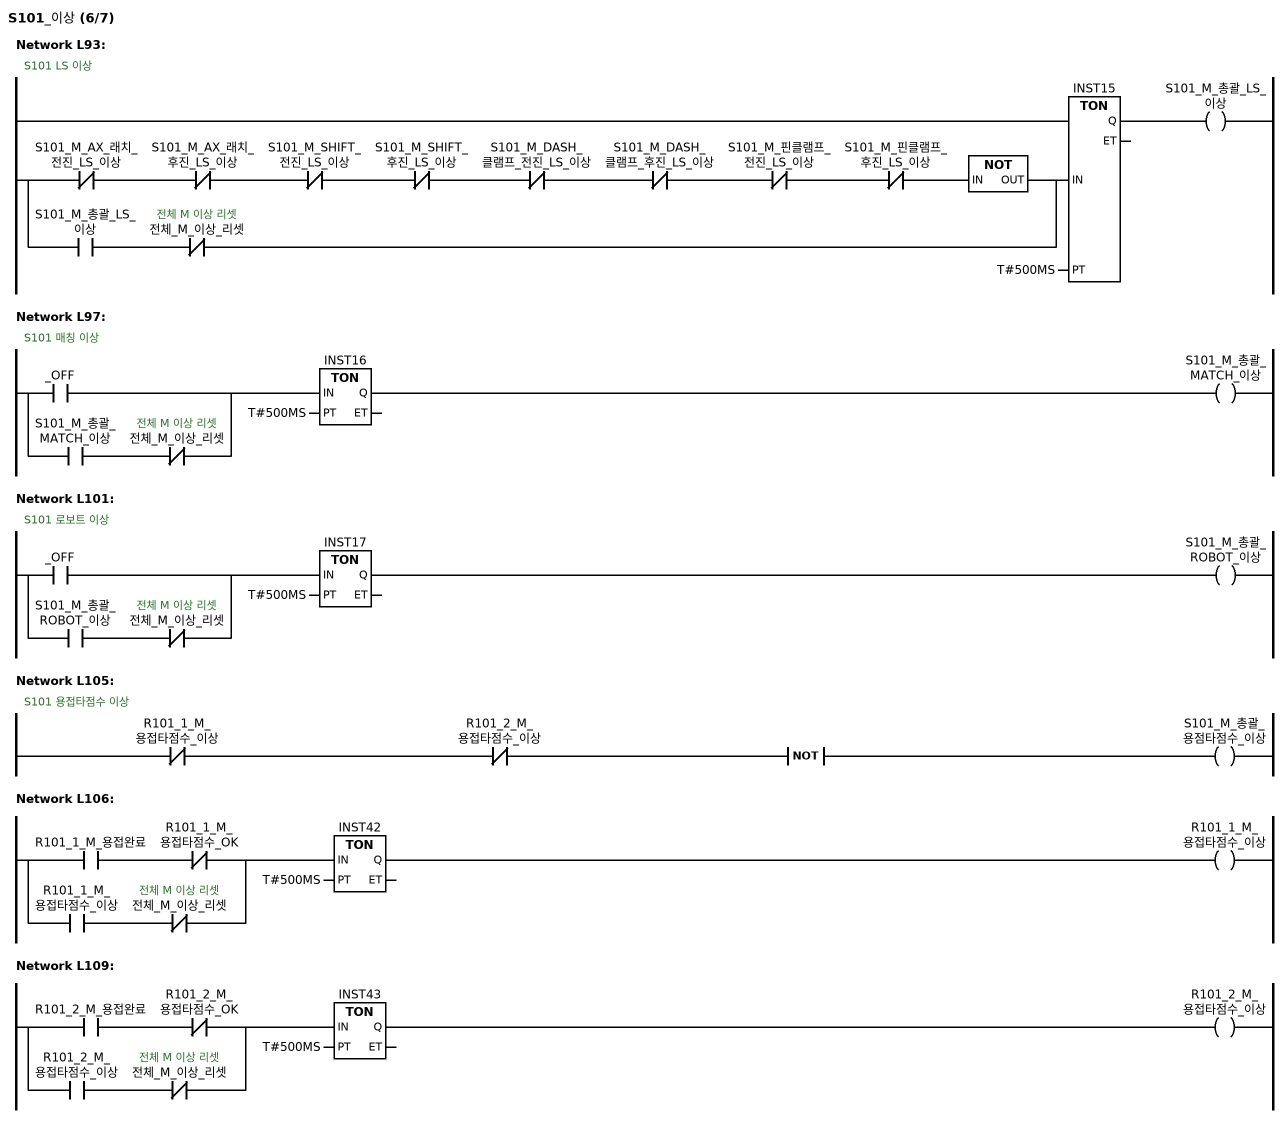
(* [picture p96: S101_이상 rungs L93-L109] *)
(* S101 LS 이상 *)
(* Rung L93 *)
INST15(IN := (NOT (NOT S101_M_AX_래치_전진_LS_이상 AND NOT S101_M_AX_래치_후진_LS_이상 AND NOT S101_M_SHIFT_전진_LS_이상 AND NOT S101_M_SHIFT_후진_LS_이상 AND NOT S101_M_DASH_클램프_전진_LS_이상 AND NOT S101_M_DASH_클램프_후진_LS_이상 AND NOT S101_M_핀클램프_전진_LS_이상 AND NOT S101_M_핀클램프_후진_LS_이상)) OR (S101_M_총괄_LS_이상 AND NOT 전체_M_이상_리셋), PT := T#500MS);
S101_M_총괄_LS_이상 := INST15.Q;
(* S101 매칭 이상 *)
(* Rung L97 *)
INST16(IN := _OFF OR (S101_M_총괄_MATCH_이상 AND NOT 전체_M_이상_리셋), PT := T#500MS);
S101_M_총괄_MATCH_이상 := INST16.Q;
(* S101 로보트 이상 *)
(* Rung L101 *)
INST17(IN := _OFF OR (S101_M_총괄_ROBOT_이상 AND NOT 전체_M_이상_리셋), PT := T#500MS);
S101_M_총괄_ROBOT_이상 := INST17.Q;
(* S101 용접타점수 이상 *)
(* Rung L105 *)
S101_M_총괄_용점타점수_이상 := NOT (NOT R101_1_M_용접타점수_이상 AND NOT R101_2_M_용접타점수_이상);
(* Rung L106 *)
INST42(IN := (R101_1_M_용접완료 AND NOT R101_1_M_용접타점수_OK) OR (R101_1_M_용접타점수_이상 AND NOT 전체_M_이상_리셋), PT := T#500MS);
R101_1_M_용접타점수_이상 := INST42.Q;
(* Rung L109 *)
INST43(IN := (R101_2_M_용접완료 AND NOT R101_2_M_용접타점수_OK) OR (R101_2_M_용접타점수_이상 AND NOT 전체_M_이상_리셋), PT := T#500MS);
R101_2_M_용접타점수_이상 := INST43.Q;

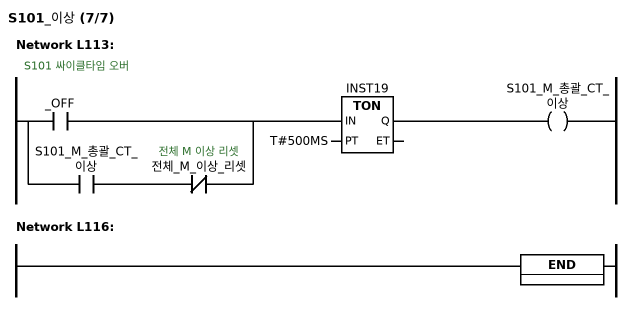
(* S101 싸이클타임 오버 *)
(* Rung L113 *)
INST19(IN := _OFF OR (S101_M_총괄_CT_이상 AND NOT 전체_M_이상_리셋), PT := T#500MS);
S101_M_총괄_CT_이상 := INST19.Q;
(* Rung L116 *)
END();
END_PROGRAM

PROGRAM S102_유틸리티 (* task: 스캔 프로그램 *)
VAR_EXTERNAL
    AWAYS_ON : BOOL; (* AT %MW3.1 *)
    MCP_PBL_102_자동_운전 : BOOL; (* AT %MW87630.7 *) (* 입력 접점 07 *)
    MCP_PBL_운전준비_ON : BOOL; (* AT %MW87630.0 *) (* 입력 접점 00 *)
    MCP_SSP_102_수동_선택 : BOOL; (* AT %MW87630.5 *) (* 입력 접점 05 *)
    MCP_SSP_102_자동_선택 : BOOL; (* AT %MW87630.6 *) (* 입력 접점 06 *)
    R102_1_1_M_I_RB_2차_작업완료 : BOOL; (* AT %MW20091.3 *)
    R102_1_1_M_I_RB_간섭무_1 : BOOL; (* AT %MW20092.0 *)
    R102_1_1_M_I_RB_원위치 : BOOL; (* AT %MW20090.3 *)
    R102_1_1_M_SEQ : WORD; (* AT %MW10040 *) (* R102_1_1_M_SEQ *)
    R102_1_1_M_STN_차종_NONE : BOOL; (* AT %MW1502.3 *)
    R102_1_1_M_STN_차종_ON : BOOL; (* AT %MW1502.2 *)
    R102_1_1_M_차종1_AX : BOOL; (* AT %MW10041.0 *) (* R102_1_1_M_차종1_AX *)
    R102_1_1_M_차종1_B : BOOL; (* AT %MW10041.1 *) (* R102_1_1_M_차종1_B *)
    R102_1_1_M_차종1_C : BOOL; (* AT %MW10041.2 *) (* R102_1_1_M_차종1_C *)
    R102_1_1_M_차종1_D : BOOL; (* AT %MW10041.3 *) (* R102_1_1_M_차종1_D *)
    R102_1_1_M_차종1_E : BOOL; (* AT %MW10041.4 *) (* R102_1_1_M_차종1_E *)
    R102_1_1_M_차종1_F : BOOL; (* AT %MW10041.5 *) (* R102_1_1_M_차종1_F *)
    R102_1_1_M_차종1_G : BOOL; (* AT %MW10041.6 *) (* R102_1_1_M_차종1_G *)
    R102_1_1_M_차종1_H : BOOL; (* AT %MW10041.7 *) (* R102_1_1_M_차종1_H *)
    R102_1_1_M_차종2_3DR : BOOL; (* AT %MW10041.8 *) (* R102_1_1_M_차종2_3DR *)
    R102_1_1_M_차종2_4DR : BOOL; (* AT %MW10041.9 *) (* R102_1_1_M_차종2_4DR *)
    R102_1_1_M_차종2_5DR : BOOL; (* AT %MW10041.10 *) (* R102_1_1_M_차종2_5DR *)
    R102_1_1_M_차종2_SP1 : BOOL; (* AT %MW10041.12 *) (* R102_1_1_M_차종2_SP1 *)
    R102_1_1_M_차종2_SP2 : BOOL; (* AT %MW10041.13 *) (* R102_1_1_M_차종2_SP2 *)
    R102_1_1_M_차종2_WGN : BOOL; (* AT %MW10041.11 *) (* R102_1_1_M_차종2_WGN *)
    R102_1_1_M_차종3_LHD : BOOL; (* AT %MW10041.14 *) (* R102_1_1_M_차종3_LHD *)
    R102_1_1_M_차종3_RHD : BOOL; (* AT %MW10041.15 *) (* R102_1_1_M_차종3_RHD *)
    R102_1_1_M_차종4_EEC : BOOL; (* AT %MW10042.3 *) (* R102_1_1_M_차종4_EEC *)
    R102_1_1_M_차종4_SP1 : BOOL; (* AT %MW10042.8 *) (* R102_1_1_M_차종4_SP1 *)
    R102_1_1_M_차종4_SP2 : BOOL; (* AT %MW10042.9 *) (* R102_1_1_M_차종4_SP2 *)
    R102_1_1_M_차종4_SP3 : BOOL; (* AT %MW10042.11 *) (* R102_1_1_M_차종4_SP3 *)
    R102_1_1_M_차종4_SP4 : BOOL; (* AT %MW10042.12 *) (* R102_1_1_M_차종4_SP4 *)
    R102_1_1_M_차종4_SP5 : BOOL; (* AT %MW10042.13 *) (* R102_1_1_M_차종4_SP5 *)
    R102_1_1_M_차종4_SP6 : BOOL; (* AT %MW10042.14 *) (* R102_1_1_M_차종4_SP6 *)
    R102_1_1_M_차종4_SP7 : BOOL; (* AT %MW10042.15 *) (* R102_1_1_M_차종4_SP7 *)
    R102_1_1_M_차종4_내수 : BOOL; (* AT %MW10042.0 *) (* R102_1_1_M_차종4_내수 *)
    R102_1_1_M_차종4_러시아 : BOOL; (* AT %MW10042.10 *) (* R102_1_1_M_차종4_러시아 *)
    R102_1_1_M_차종4_북미 : BOOL; (* AT %MW10042.2 *) (* R102_1_1_M_차종4_북미 *)
    R102_1_1_M_차종4_브라질 : BOOL; (* AT %MW10042.7 *) (* R102_1_1_M_차종4_브라질 *)
    R102_1_1_M_차종4_수출 : BOOL; (* AT %MW10042.1 *) (* R102_1_1_M_차종4_수출 *)
    R102_1_1_M_차종4_중국 : BOOL; (* AT %MW10042.6 *) (* R102_1_1_M_차종4_중국 *)
    R102_1_1_M_차종4_중동 : BOOL; (* AT %MW10042.5 *) (* R102_1_1_M_차종4_중동 *)
    R102_1_1_M_차종4_호주 : BOOL; (* AT %MW10042.4 *) (* R102_1_1_M_차종4_호주 *)
    R102_1_1_M_차종5_AT : BOOL; (* AT %MW10043.1 *) (* R102_1_1_M_차종5_AT *)
    R102_1_1_M_차종5_MT : BOOL; (* AT %MW10043.0 *) (* R102_1_1_M_차종5_MT *)
    R102_1_1_M_차종5_SP1 : BOOL; (* AT %MW10043.2 *) (* R102_1_1_M_차종5_SP1 *)
    R102_1_1_M_차종6_DSROOF : BOOL; (* AT %MW10043.6 *) (* R102_1_1_M_차종6_DSROOF *)
    R102_1_1_M_차종6_SP1 : BOOL; (* AT %MW10043.7 *) (* R102_1_1_M_차종6_SP1 *)
    R102_1_1_M_차종6_썬루프 : BOOL; (* AT %MW10043.4 *) (* R102_1_1_M_차종6_썬루프 *)
    R102_1_1_M_차종6_일반루프 : BOOL; (* AT %MW10043.3 *) (* R102_1_1_M_차종6_일반루프 *)
    R102_1_1_M_차종6_파노라마루프 : BOOL; (* AT %MW10043.5 *) (* R102_1_1_M_차종6_파노라마루프 *)
    R102_1_1_M_차종7_DSL : BOOL; (* AT %MW10043.9 *) (* R102_1_1_M_차종7_DSL *)
    R102_1_1_M_차종7_GSL : BOOL; (* AT %MW10043.8 *) (* R102_1_1_M_차종7_GSL *)
    R102_1_1_M_차종7_SP1 : BOOL; (* AT %MW10043.10 *) (* R102_1_1_M_차종7_SP1 *)
    R102_1_1_M_차종7_SP2 : BOOL; (* AT %MW10043.11 *) (* R102_1_1_M_차종7_SP2 *)
    R102_1_1_M_차종7_SP3 : BOOL; (* AT %MW10043.12 *) (* R102_1_1_M_차종7_SP3 *)
    R102_1_1_M_차종7_SP4 : BOOL; (* AT %MW10043.13 *) (* R102_1_1_M_차종7_SP4 *)
    R102_1_1_M_차종7_SP5 : BOOL; (* AT %MW10043.14 *) (* R102_1_1_M_차종7_SP5 *)
    R102_1_1_M_차종7_SP6 : BOOL; (* AT %MW10043.15 *) (* R102_1_1_M_차종7_SP6 *)
    R102_1_1_M_차종8_2WD : BOOL; (* AT %MW10044.0 *) (* R102_1_1_M_차종8_2WD *)
    R102_1_1_M_차종8_4WD : BOOL; (* AT %MW10044.1 *) (* R102_1_1_M_차종8_4WD *)
    R102_1_1_M_차종8_SP1 : BOOL; (* AT %MW10044.2 *) (* R102_1_1_M_차종8_SP1 *)
    R102_1_1_M_차종9_MPI : BOOL; (* AT %MW10044.3 *) (* R102_1_1_M_차종9_MPI *)
    R102_1_1_M_차종9_SP1 : BOOL; (* AT %MW10044.5 *) (* R102_1_1_M_차종9_SP1 *)
    R102_1_1_M_차종9_SP10 : BOOL; (* AT %MW10044.14 *) (* R102_1_1_M_차종9_SP10 *)
    R102_1_1_M_차종9_SP11 : BOOL; (* AT %MW10044.15 *) (* R102_1_1_M_차종9_SP11 *)
    R102_1_1_M_차종9_SP2 : BOOL; (* AT %MW10044.6 *) (* R102_1_1_M_차종9_SP2 *)
    R102_1_1_M_차종9_SP3 : BOOL; (* AT %MW10044.7 *) (* R102_1_1_M_차종9_SP3 *)
    R102_1_1_M_차종9_SP4 : BOOL; (* AT %MW10044.8 *) (* R102_1_1_M_차종9_SP4 *)
    R102_1_1_M_차종9_SP5 : BOOL; (* AT %MW10044.9 *) (* R102_1_1_M_차종9_SP5 *)
    R102_1_1_M_차종9_SP6 : BOOL; (* AT %MW10044.10 *) (* R102_1_1_M_차종9_SP6 *)
    R102_1_1_M_차종9_SP7 : BOOL; (* AT %MW10044.11 *) (* R102_1_1_M_차종9_SP7 *)
    R102_1_1_M_차종9_SP8 : BOOL; (* AT %MW10044.12 *) (* R102_1_1_M_차종9_SP8 *)
    R102_1_1_M_차종9_SP9 : BOOL; (* AT %MW10044.13 *) (* R102_1_1_M_차종9_SP9 *)
    R102_1_1_M_차종9_T_GDI : BOOL; (* AT %MW10044.4 *) (* R102_1_1_M_차종9_T_GDI *)
    R102_1_1_M_차종_OPT1_R_RACK_무 : BOOL; (* AT %MW10045.3 *) (* R102_1_1_M_차종_OPT1_R_RACK_무 *)
    R102_1_1_M_차종_OPT1_R_RACK_유 : BOOL; (* AT %MW10045.2 *) (* R102_1_1_M_차종_OPT1_R_RACK_유 *)
    R102_1_1_M_차종_OPT1_SP1 : BOOL; (* AT %MW10045.10 *) (* R102_1_1_M_차종_OPT1_SP1 *)
    R102_1_1_M_차종_OPT1_SP2 : BOOL; (* AT %MW10045.11 *) (* R102_1_1_M_차종_OPT1_SP2 *)
    R102_1_1_M_차종_OPT1_SP3 : BOOL; (* AT %MW10045.12 *) (* R102_1_1_M_차종_OPT1_SP3 *)
    R102_1_1_M_차종_OPT1_SP4 : BOOL; (* AT %MW10045.13 *) (* R102_1_1_M_차종_OPT1_SP4 *)
    R102_1_1_M_차종_OPT1_SP5 : BOOL; (* AT %MW10045.14 *) (* R102_1_1_M_차종_OPT1_SP5 *)
    R102_1_1_M_차종_OPT1_SP6 : BOOL; (* AT %MW10045.15 *) (* R102_1_1_M_차종_OPT1_SP6 *)
    R102_1_1_M_차종_OPT1_S_REP_EATER_무 : BOOL; (* AT %MW10045.7 *) (* R102_1_1_M_차종_OPT1_S_REP_EATER_무 *)
    R102_1_1_M_차종_OPT1_S_REP_EATER_유 : BOOL; (* AT %MW10045.6 *) (* R102_1_1_M_차종_OPT1_S_REP_EATER_유 *)
    R102_1_1_M_차종_OPT1_VAN_무 : BOOL; (* AT %MW10045.9 *) (* R102_1_1_M_차종_OPT1_VAN_무 *)
    R102_1_1_M_차종_OPT1_VAN_유 : BOOL; (* AT %MW10045.8 *) (* R102_1_1_M_차종_OPT1_VAN_유 *)
    R102_1_1_M_차종_OPT1_슬라이딩_무 : BOOL; (* AT %MW10045.1 *) (* R102_1_1_M_차종_OPT1_슬라이딩_무 *)
    R102_1_1_M_차종_OPT1_슬라이딩_유 : BOOL; (* AT %MW10045.0 *) (* R102_1_1_M_차종_OPT1_슬라이딩_유 *)
    R102_1_1_M_차종_OPT1_폴딩_무 : BOOL; (* AT %MW10045.5 *) (* R102_1_1_M_차종_OPT1_폴딩_무 *)
    R102_1_1_M_차종_OPT1_폴딩_유 : BOOL; (* AT %MW10045.4 *) (* R102_1_1_M_차종_OPT1_폴딩_유 *)
    R102_1_M_I_RB_간섭무_1 : BOOL; (* AT %MW20082.0 *)
    R102_1_M_I_RB_원위치 : BOOL; (* AT %MW20080.3 *)
    R102_1_M_SEQ : WORD; (* AT %MW10080 *) (* R102_1_M_SEQ *)
    R102_1_M_STN_차종_NONE : BOOL; (* AT %MW1502.5 *)
    R102_1_M_STN_차종_ON : BOOL; (* AT %MW1502.4 *)
    R102_1_M_차종1_AX : BOOL; (* AT %MW10081.0 *) (* R102_1_M_차종1_AX *)
    R102_1_M_차종1_B : BOOL; (* AT %MW10081.1 *) (* R102_1_M_차종1_B *)
    R102_1_M_차종1_C : BOOL; (* AT %MW10081.2 *) (* R102_1_M_차종1_C *)
    R102_1_M_차종1_D : BOOL; (* AT %MW10081.3 *) (* R102_1_M_차종1_D *)
    R102_1_M_차종1_E : BOOL; (* AT %MW10081.4 *) (* R102_1_M_차종1_E *)
    R102_1_M_차종1_F : BOOL; (* AT %MW10081.5 *) (* R102_1_M_차종1_F *)
    R102_1_M_차종1_G : BOOL; (* AT %MW10081.6 *) (* R102_1_M_차종1_G *)
    R102_1_M_차종1_H : BOOL; (* AT %MW10081.7 *) (* R102_1_M_차종1_H *)
    R102_1_M_차종2_3DR : BOOL; (* AT %MW10081.8 *) (* R102_1_M_차종2_3DR *)
    R102_1_M_차종2_4DR : BOOL; (* AT %MW10081.9 *) (* R102_1_M_차종2_4DR *)
    R102_1_M_차종2_5DR : BOOL; (* AT %MW10081.10 *) (* R102_1_M_차종2_5DR *)
    R102_1_M_차종2_SP1 : BOOL; (* AT %MW10081.12 *) (* R102_1_M_차종2_SP1 *)
    R102_1_M_차종2_SP2 : BOOL; (* AT %MW10081.13 *) (* R102_1_M_차종2_SP2 *)
    R102_1_M_차종2_WGN : BOOL; (* AT %MW10081.11 *) (* R102_1_M_차종2_WGN *)
    R102_1_M_차종3_LHD : BOOL; (* AT %MW10081.14 *) (* R102_1_M_차종3_LHD *)
    R102_1_M_차종3_RHD : BOOL; (* AT %MW10081.15 *) (* R102_1_M_차종3_RHD *)
    R102_1_M_차종4_EEC : BOOL; (* AT %MW10082.3 *) (* R102_1_M_차종4_EEC *)
    R102_1_M_차종4_SP1 : BOOL; (* AT %MW10082.8 *) (* R102_1_M_차종4_SP1 *)
    R102_1_M_차종4_SP2 : BOOL; (* AT %MW10082.9 *) (* R102_1_M_차종4_SP2 *)
    R102_1_M_차종4_SP3 : BOOL; (* AT %MW10082.11 *) (* R102_1_M_차종4_SP3 *)
    R102_1_M_차종4_SP4 : BOOL; (* AT %MW10082.12 *) (* R102_1_M_차종4_SP4 *)
    R102_1_M_차종4_SP5 : BOOL; (* AT %MW10082.13 *) (* R102_1_M_차종4_SP5 *)
    R102_1_M_차종4_SP6 : BOOL; (* AT %MW10082.14 *) (* R102_1_M_차종4_SP6 *)
    R102_1_M_차종4_SP7 : BOOL; (* AT %MW10082.15 *) (* R102_1_M_차종4_SP7 *)
    R102_1_M_차종4_내수 : BOOL; (* AT %MW10082.0 *) (* R102_1_M_차종4_내수 *)
    R102_1_M_차종4_러시아 : BOOL; (* AT %MW10082.10 *) (* R102_1_M_차종4_러시아 *)
    R102_1_M_차종4_북미 : BOOL; (* AT %MW10082.2 *) (* R102_1_M_차종4_북미 *)
    R102_1_M_차종4_브라질 : BOOL; (* AT %MW10082.7 *) (* R102_1_M_차종4_브라질 *)
    R102_1_M_차종4_수출 : BOOL; (* AT %MW10082.1 *) (* R102_1_M_차종4_수출 *)
    R102_1_M_차종4_중국 : BOOL; (* AT %MW10082.6 *) (* R102_1_M_차종4_중국 *)
    R102_1_M_차종4_중동 : BOOL; (* AT %MW10082.5 *) (* R102_1_M_차종4_중동 *)
    R102_1_M_차종4_호주 : BOOL; (* AT %MW10082.4 *) (* R102_1_M_차종4_호주 *)
    R102_1_M_차종5_AT : BOOL; (* AT %MW10083.1 *) (* R102_1_M_차종5_AT *)
    R102_1_M_차종5_MT : BOOL; (* AT %MW10083.0 *) (* R102_1_M_차종5_MT *)
    R102_1_M_차종5_SP1 : BOOL; (* AT %MW10083.2 *) (* R102_1_M_차종5_SP1 *)
    R102_1_M_차종6_DSROOF : BOOL; (* AT %MW10083.6 *) (* R102_1_M_차종6_DSROOF *)
    R102_1_M_차종6_SP1 : BOOL; (* AT %MW10083.7 *) (* R102_1_M_차종6_SP1 *)
    R102_1_M_차종6_썬루프 : BOOL; (* AT %MW10083.4 *) (* R102_1_M_차종6_썬루프 *)
    R102_1_M_차종6_일반루프 : BOOL; (* AT %MW10083.3 *) (* R102_1_M_차종6_일반루프 *)
    R102_1_M_차종6_파노라마루프 : BOOL; (* AT %MW10083.5 *) (* R102_1_M_차종6_파노라마루프 *)
    R102_1_M_차종7_DSL : BOOL; (* AT %MW10083.9 *) (* R102_1_M_차종7_DSL *)
    R102_1_M_차종7_GSL : BOOL; (* AT %MW10083.8 *) (* R102_1_M_차종7_GSL *)
    R102_1_M_차종7_SP1 : BOOL; (* AT %MW10083.10 *) (* R102_1_M_차종7_SP1 *)
    R102_1_M_차종7_SP2 : BOOL; (* AT %MW10083.11 *) (* R102_1_M_차종7_SP2 *)
    R102_1_M_차종7_SP3 : BOOL; (* AT %MW10083.12 *) (* R102_1_M_차종7_SP3 *)
    R102_1_M_차종7_SP4 : BOOL; (* AT %MW10083.13 *) (* R102_1_M_차종7_SP4 *)
    R102_1_M_차종7_SP5 : BOOL; (* AT %MW10083.14 *) (* R102_1_M_차종7_SP5 *)
    R102_1_M_차종7_SP6 : BOOL; (* AT %MW10083.15 *) (* R102_1_M_차종7_SP6 *)
    R102_1_M_차종8_2WD : BOOL; (* AT %MW10084.0 *) (* R102_1_M_차종8_2WD *)
    R102_1_M_차종8_4WD : BOOL; (* AT %MW10084.1 *) (* R102_1_M_차종8_4WD *)
    R102_1_M_차종8_SP1 : BOOL; (* AT %MW10084.2 *) (* R102_1_M_차종8_SP1 *)
    R102_1_M_차종9_MPI : BOOL; (* AT %MW10084.3 *) (* R102_1_M_차종9_MPI *)
    R102_1_M_차종9_SP1 : BOOL; (* AT %MW10084.5 *) (* R102_1_M_차종9_SP1 *)
    R102_1_M_차종9_SP10 : BOOL; (* AT %MW10084.14 *) (* R102_1_M_차종9_SP10 *)
    R102_1_M_차종9_SP11 : BOOL; (* AT %MW10084.15 *) (* R102_1_M_차종9_SP11 *)
    R102_1_M_차종9_SP2 : BOOL; (* AT %MW10084.6 *) (* R102_1_M_차종9_SP2 *)
    R102_1_M_차종9_SP3 : BOOL; (* AT %MW10084.7 *) (* R102_1_M_차종9_SP3 *)
    R102_1_M_차종9_SP4 : BOOL; (* AT %MW10084.8 *) (* R102_1_M_차종9_SP4 *)
    R102_1_M_차종9_SP5 : BOOL; (* AT %MW10084.9 *) (* R102_1_M_차종9_SP5 *)
    R102_1_M_차종9_SP6 : BOOL; (* AT %MW10084.10 *) (* R102_1_M_차종9_SP6 *)
    R102_1_M_차종9_SP7 : BOOL; (* AT %MW10084.11 *) (* R102_1_M_차종9_SP7 *)
    R102_1_M_차종9_SP8 : BOOL; (* AT %MW10084.12 *) (* R102_1_M_차종9_SP8 *)
    R102_1_M_차종9_SP9 : BOOL; (* AT %MW10084.13 *) (* R102_1_M_차종9_SP9 *)
    R102_1_M_차종9_T_GDI : BOOL; (* AT %MW10084.4 *) (* R102_1_M_차종9_T_GDI *)
    R102_1_M_차종_OPT1_R_RACK_무 : BOOL; (* AT %MW10085.3 *) (* R102_1_M_차종_OPT1_R_RACK_무 *)
    R102_1_M_차종_OPT1_R_RACK_유 : BOOL; (* AT %MW10085.2 *) (* R102_1_M_차종_OPT1_R_RACK_유 *)
    R102_1_M_차종_OPT1_SP1 : BOOL; (* AT %MW10085.10 *) (* R102_1_M_차종_OPT1_SP1 *)
    R102_1_M_차종_OPT1_SP2 : BOOL; (* AT %MW10085.11 *) (* R102_1_M_차종_OPT1_SP2 *)
    R102_1_M_차종_OPT1_SP3 : BOOL; (* AT %MW10085.12 *) (* R102_1_M_차종_OPT1_SP3 *)
    R102_1_M_차종_OPT1_SP4 : BOOL; (* AT %MW10085.13 *) (* R102_1_M_차종_OPT1_SP4 *)
    R102_1_M_차종_OPT1_SP5 : BOOL; (* AT %MW10085.14 *) (* R102_1_M_차종_OPT1_SP5 *)
    R102_1_M_차종_OPT1_SP6 : BOOL; (* AT %MW10085.15 *) (* R102_1_M_차종_OPT1_SP6 *)
    R102_1_M_차종_OPT1_S_REP_EATER_무 : BOOL; (* AT %MW10085.7 *) (* R102_1_M_차종_OPT1_S_REP_EATER_무 *)
    R102_1_M_차종_OPT1_S_REP_EATER_유 : BOOL; (* AT %MW10085.6 *) (* R102_1_M_차종_OPT1_S_REP_EATER_유 *)
    R102_1_M_차종_OPT1_VAN_무 : BOOL; (* AT %MW10085.9 *) (* R102_1_M_차종_OPT1_VAN_무 *)
    R102_1_M_차종_OPT1_VAN_유 : BOOL; (* AT %MW10085.8 *) (* R102_1_M_차종_OPT1_VAN_유 *)
    R102_1_M_차종_OPT1_슬라이딩_무 : BOOL; (* AT %MW10085.1 *) (* R102_1_M_차종_OPT1_슬라이딩_무 *)
    R102_1_M_차종_OPT1_슬라이딩_유 : BOOL; (* AT %MW10085.0 *) (* R102_1_M_차종_OPT1_슬라이딩_유 *)
    R102_1_M_차종_OPT1_폴딩_무 : BOOL; (* AT %MW10085.5 *) (* R102_1_M_차종_OPT1_폴딩_무 *)
    R102_1_M_차종_OPT1_폴딩_유 : BOOL; (* AT %MW10085.4 *) (* R102_1_M_차종_OPT1_폴딩_유 *)
    S102_M_SEQ : WORD; (* AT %MW10060 *) (* S102_M_SEQ *)
    S102_M_STN_DASH_로딩완료 : BOOL; (* AT %MW1501.8 *)
    S102_M_STN_차종_NONE : BOOL; (* AT %MW1502.1 *)
    S102_M_STN_차종_ON : BOOL; (* AT %MW1502.0 *)
    S102_M_공정_HOME_POSI : BOOL; (* AT %MW1504.0 *)
    S102_M_공정_간섭무 : BOOL; (* AT %MW1504.1 *)
    S102_M_공정_사양감지_OK : BOOL; (* AT %MW1501.5 *)
    S102_M_공정_제품감지_OFF : BOOL; (* AT %MW1501.4 *)
    S102_M_공정_제품감지_ON : BOOL; (* AT %MW1501.3 *)
    S102_M_사양_이상 : BOOL; (* AT %MW1516.0 *)
    S102_M_수동_모드 : BOOL; (* AT %MW1500.3 *)
    S102_M_운전준비_ON : BOOL; (* AT %MW1500.0 *)
    S102_M_자동_START : BOOL; (* AT %MW1500.5 *)
    S102_M_자동_모드 : BOOL; (* AT %MW1500.1 *)
    S102_M_자동_운전중 : BOOL; (* AT %MW1500.4 *)
    S102_M_작업_완료 : BOOL; (* AT %MW1501.0 *)
    S102_M_작업_완료_보조 : BOOL; (* AT %MW1500.9 *)
    S102_M_차종1_AX : BOOL; (* AT %MW10061.0 *) (* S102_M_차종1_AX *)
    S102_M_차종1_B : BOOL; (* AT %MW10061.1 *) (* S102_M_차종1_B *)
    S102_M_차종1_C : BOOL; (* AT %MW10061.2 *) (* S102_M_차종1_C *)
    S102_M_차종1_D : BOOL; (* AT %MW10061.3 *) (* S102_M_차종1_D *)
    S102_M_차종1_E : BOOL; (* AT %MW10061.4 *) (* S102_M_차종1_E *)
    S102_M_차종1_F : BOOL; (* AT %MW10061.5 *) (* S102_M_차종1_F *)
    S102_M_차종1_G : BOOL; (* AT %MW10061.6 *) (* S102_M_차종1_G *)
    S102_M_차종1_H : BOOL; (* AT %MW10061.7 *) (* S102_M_차종1_H *)
    S102_M_차종2_3DR : BOOL; (* AT %MW10061.8 *) (* S102_M_차종2_3DR *)
    S102_M_차종2_4DR : BOOL; (* AT %MW10061.9 *) (* S102_M_차종2_4DR *)
    S102_M_차종2_5DR : BOOL; (* AT %MW10061.10 *) (* S102_M_차종2_5DR *)
    S102_M_차종2_SP1 : BOOL; (* AT %MW10061.12 *) (* S102_M_차종2_SP1 *)
    S102_M_차종2_SP2 : BOOL; (* AT %MW10061.13 *) (* S102_M_차종2_SP2 *)
    S102_M_차종2_WGN : BOOL; (* AT %MW10061.11 *) (* S102_M_차종2_WGN *)
    S102_M_차종3_LHD : BOOL; (* AT %MW10061.14 *) (* S102_M_차종3_LHD *)
    S102_M_차종3_RHD : BOOL; (* AT %MW10061.15 *) (* S102_M_차종3_RHD *)
    S102_M_차종4_EEC : BOOL; (* AT %MW10062.3 *) (* S102_M_차종4_EEC *)
    S102_M_차종4_SP1 : BOOL; (* AT %MW10062.8 *) (* S102_M_차종4_SP1 *)
    S102_M_차종4_SP2 : BOOL; (* AT %MW10062.9 *) (* S102_M_차종4_SP2 *)
    S102_M_차종4_SP3 : BOOL; (* AT %MW10062.11 *) (* S102_M_차종4_SP3 *)
    S102_M_차종4_SP4 : BOOL; (* AT %MW10062.12 *) (* S102_M_차종4_SP4 *)
    S102_M_차종4_SP5 : BOOL; (* AT %MW10062.13 *) (* S102_M_차종4_SP5 *)
    S102_M_차종4_SP6 : BOOL; (* AT %MW10062.14 *) (* S102_M_차종4_SP6 *)
    S102_M_차종4_SP7 : BOOL; (* AT %MW10062.15 *) (* S102_M_차종4_SP7 *)
    S102_M_차종4_내수 : BOOL; (* AT %MW10062.0 *) (* S102_M_차종4_내수 *)
    S102_M_차종4_러시아 : BOOL; (* AT %MW10062.10 *) (* S102_M_차종4_러시아 *)
    S102_M_차종4_북미 : BOOL; (* AT %MW10062.2 *) (* S102_M_차종4_북미 *)
    S102_M_차종4_브라질 : BOOL; (* AT %MW10062.7 *) (* S102_M_차종4_브라질 *)
    S102_M_차종4_수출 : BOOL; (* AT %MW10062.1 *) (* S102_M_차종4_수출 *)
    S102_M_차종4_중국 : BOOL; (* AT %MW10062.6 *) (* S102_M_차종4_중국 *)
    S102_M_차종4_중동 : BOOL; (* AT %MW10062.5 *) (* S102_M_차종4_중동 *)
    S102_M_차종4_호주 : BOOL; (* AT %MW10062.4 *) (* S102_M_차종4_호주 *)
    S102_M_차종5_AT : BOOL; (* AT %MW10063.1 *) (* S102_M_차종5_AT *)
    S102_M_차종5_MT : BOOL; (* AT %MW10063.0 *) (* S102_M_차종5_MT *)
    S102_M_차종5_SP1 : BOOL; (* AT %MW10063.2 *) (* S102_M_차종5_SP1 *)
    S102_M_차종6_DSROOF : BOOL; (* AT %MW10063.6 *) (* S102_M_차종6_DSROOF *)
    S102_M_차종6_SP1 : BOOL; (* AT %MW10063.7 *) (* S102_M_차종6_SP1 *)
    S102_M_차종6_썬루프 : BOOL; (* AT %MW10063.4 *) (* S102_M_차종6_썬루프 *)
    S102_M_차종6_일반루프 : BOOL; (* AT %MW10063.3 *) (* S102_M_차종6_일반루프 *)
    S102_M_차종6_파노라마루프 : BOOL; (* AT %MW10063.5 *) (* S102_M_차종6_파노라마루프 *)
    S102_M_차종7_DSL : BOOL; (* AT %MW10063.9 *) (* S102_M_차종7_DSL *)
    S102_M_차종7_GSL : BOOL; (* AT %MW10063.8 *) (* S102_M_차종7_GSL *)
    S102_M_차종7_SP1 : BOOL; (* AT %MW10063.10 *) (* S102_M_차종7_SP1 *)
    S102_M_차종7_SP2 : BOOL; (* AT %MW10063.11 *) (* S102_M_차종7_SP2 *)
    S102_M_차종7_SP3 : BOOL; (* AT %MW10063.12 *) (* S102_M_차종7_SP3 *)
    S102_M_차종7_SP4 : BOOL; (* AT %MW10063.13 *) (* S102_M_차종7_SP4 *)
    S102_M_차종7_SP5 : BOOL; (* AT %MW10063.14 *) (* S102_M_차종7_SP5 *)
    S102_M_차종7_SP6 : BOOL; (* AT %MW10063.15 *) (* S102_M_차종7_SP6 *)
    S102_M_차종8_2WD : BOOL; (* AT %MW10064.0 *) (* S102_M_차종8_2WD *)
    S102_M_차종8_4WD : BOOL; (* AT %MW10064.1 *) (* S102_M_차종8_4WD *)
    S102_M_차종8_SP1 : BOOL; (* AT %MW10064.2 *) (* S102_M_차종8_SP1 *)
    S102_M_차종9_MPI : BOOL; (* AT %MW10064.3 *) (* S102_M_차종9_MPI *)
    S102_M_차종9_SP1 : BOOL; (* AT %MW10064.5 *) (* S102_M_차종9_SP1 *)
    S102_M_차종9_SP10 : BOOL; (* AT %MW10064.14 *) (* S102_M_차종9_SP10 *)
    S102_M_차종9_SP11 : BOOL; (* AT %MW10064.15 *) (* S102_M_차종9_SP11 *)
    S102_M_차종9_SP2 : BOOL; (* AT %MW10064.6 *) (* S102_M_차종9_SP2 *)
    S102_M_차종9_SP3 : BOOL; (* AT %MW10064.7 *) (* S102_M_차종9_SP3 *)
    S102_M_차종9_SP4 : BOOL; (* AT %MW10064.8 *) (* S102_M_차종9_SP4 *)
    S102_M_차종9_SP5 : BOOL; (* AT %MW10064.9 *) (* S102_M_차종9_SP5 *)
    S102_M_차종9_SP6 : BOOL; (* AT %MW10064.10 *) (* S102_M_차종9_SP6 *)
    S102_M_차종9_SP7 : BOOL; (* AT %MW10064.11 *) (* S102_M_차종9_SP7 *)
    S102_M_차종9_SP8 : BOOL; (* AT %MW10064.12 *) (* S102_M_차종9_SP8 *)
    S102_M_차종9_SP9 : BOOL; (* AT %MW10064.13 *) (* S102_M_차종9_SP9 *)
    S102_M_차종9_T_GDI : BOOL; (* AT %MW10064.4 *) (* S102_M_차종9_T_GDI *)
    S102_M_차종_OPT1_R_RACK_무 : BOOL; (* AT %MW10065.3 *) (* S102_M_차종_OPT1_R_RACK_무 *)
    S102_M_차종_OPT1_R_RACK_유 : BOOL; (* AT %MW10065.2 *) (* S102_M_차종_OPT1_R_RACK_유 *)
    S102_M_차종_OPT1_SP1 : BOOL; (* AT %MW10065.10 *) (* S102_M_차종_OPT1_SP1 *)
    S102_M_차종_OPT1_SP2 : BOOL; (* AT %MW10065.11 *) (* S102_M_차종_OPT1_SP2 *)
    S102_M_차종_OPT1_SP3 : BOOL; (* AT %MW10065.12 *) (* S102_M_차종_OPT1_SP3 *)
    S102_M_차종_OPT1_SP4 : BOOL; (* AT %MW10065.13 *) (* S102_M_차종_OPT1_SP4 *)
    S102_M_차종_OPT1_SP5 : BOOL; (* AT %MW10065.14 *) (* S102_M_차종_OPT1_SP5 *)
    S102_M_차종_OPT1_SP6 : BOOL; (* AT %MW10065.15 *) (* S102_M_차종_OPT1_SP6 *)
    S102_M_차종_OPT1_S_REP_EATER_무 : BOOL; (* AT %MW10065.7 *) (* S102_M_차종_OPT1_S_REP_EATER_무 *)
    S102_M_차종_OPT1_S_REP_EATER_유 : BOOL; (* AT %MW10065.6 *) (* S102_M_차종_OPT1_S_REP_EATER_유 *)
    S102_M_차종_OPT1_VAN_무 : BOOL; (* AT %MW10065.9 *) (* S102_M_차종_OPT1_VAN_무 *)
    S102_M_차종_OPT1_VAN_유 : BOOL; (* AT %MW10065.8 *) (* S102_M_차종_OPT1_VAN_유 *)
    S102_M_차종_OPT1_슬라이딩_무 : BOOL; (* AT %MW10065.1 *) (* S102_M_차종_OPT1_슬라이딩_무 *)
    S102_M_차종_OPT1_슬라이딩_유 : BOOL; (* AT %MW10065.0 *) (* S102_M_차종_OPT1_슬라이딩_유 *)
    S102_M_차종_OPT1_폴딩_무 : BOOL; (* AT %MW10065.5 *) (* S102_M_차종_OPT1_폴딩_무 *)
    S102_M_차종_OPT1_폴딩_유 : BOOL; (* AT %MW10065.4 *) (* S102_M_차종_OPT1_폴딩_유 *)
    S102_PRS_I_AT_감지 : BOOL; (* AT %MW86201.8 *)
    S102_PRS_I_AX_파트_ON : BOOL; (* AT %MW86200.1 *)
    S102_PRS_I_LHD_감지 : BOOL; (* AT %MW86201.0 *)
    S102_PRS_I_MT_감지 : BOOL; (* AT %MW86201.9 *)
    S102_PRS_I_RHD_감지 : BOOL; (* AT %MW86201.1 *)
    S102_PRS_I_공용_파트_ON : BOOL; (* AT %MW86200.0 *)
    S102_운전준비 : TON;
    T102_자동 : TON;
    전체_M_GATE_자동기동 : BOOL; (* AT %MW308.1 *) (* 전체 M GATE 자동기동 *)
    전체_라인_M_총괄_SAFETY_이상 : BOOL; (* AT %MW300.2 *)
    전체_라인_M_총괄_공기압_이상 : BOOL; (* AT %MW300.3 *)
    전체_라인_M_총괄_비상정지_이상 : BOOL; (* AT %MW300.1 *)
    전체_라인_M_총괄_이상 : BOOL; (* AT %MW300.0 *)
END_VAR
VAR
    INST : TON;
END_VAR
VAR
    _t1 : BOOL;
    _t2 : BOOL;
    _t3 : BOOL;
END_VAR

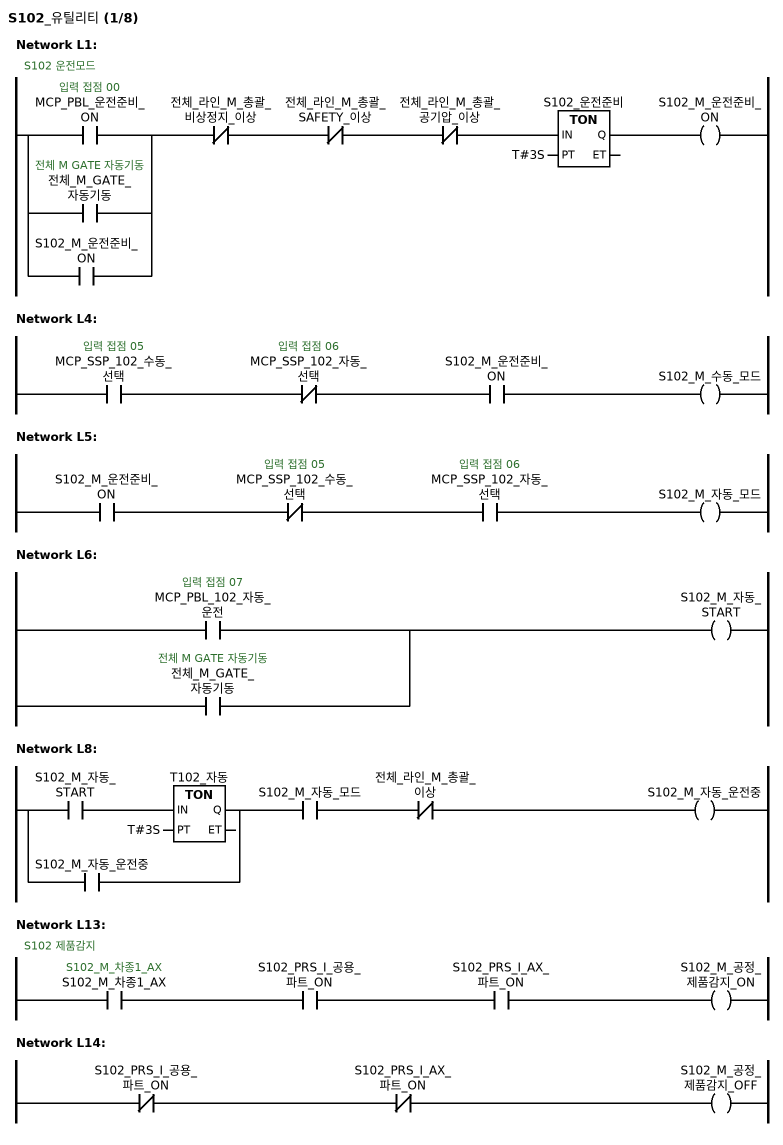
(* S102 운전모드 *)
(* Rung L1 *)
S102_운전준비(IN := (MCP_PBL_운전준비_ON OR 전체_M_GATE_자동기동 OR S102_M_운전준비_ON) AND NOT 전체_라인_M_총괄_비상정지_이상 AND NOT 전체_라인_M_총괄_SAFETY_이상 AND NOT 전체_라인_M_총괄_공기압_이상, PT := T#3S);
S102_M_운전준비_ON := S102_운전준비.Q;
(* Rung L4 *)
S102_M_수동_모드 := MCP_SSP_102_수동_선택 AND NOT MCP_SSP_102_자동_선택 AND S102_M_운전준비_ON;
(* Rung L5 *)
S102_M_자동_모드 := S102_M_운전준비_ON AND NOT MCP_SSP_102_수동_선택 AND MCP_SSP_102_자동_선택;
(* Rung L6 *)
S102_M_자동_START := MCP_PBL_102_자동_운전 OR 전체_M_GATE_자동기동;
(* Rung L8 *)
T102_자동(IN := S102_M_자동_START, PT := T#3S);
S102_M_자동_운전중 := (T102_자동.Q OR S102_M_자동_운전중) AND S102_M_자동_모드 AND NOT 전체_라인_M_총괄_이상;
(* S102 제품감지 *)
(* Rung L13 *)
S102_M_공정_제품감지_ON := S102_M_차종1_AX AND S102_PRS_I_공용_파트_ON AND S102_PRS_I_AX_파트_ON;
(* Rung L14 *)
S102_M_공정_제품감지_OFF := NOT S102_PRS_I_공용_파트_ON AND NOT S102_PRS_I_AX_파트_ON;

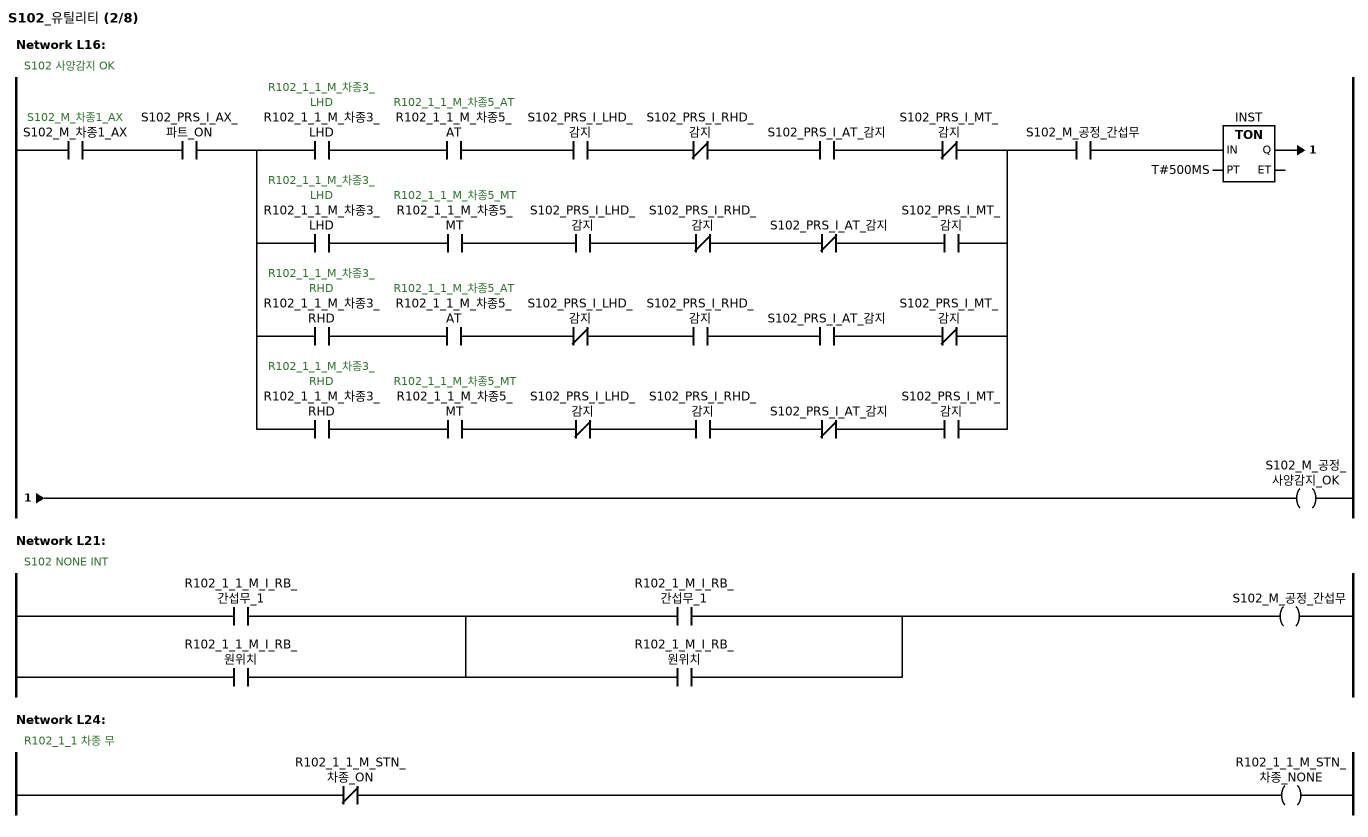
(* S102 사양감지 OK *)
(* Rung L16 *)
INST(IN := S102_M_차종1_AX AND S102_PRS_I_AX_파트_ON AND ((R102_1_1_M_차종3_LHD AND R102_1_1_M_차종5_AT AND S102_PRS_I_LHD_감지 AND NOT S102_PRS_I_RHD_감지 AND S102_PRS_I_AT_감지 AND NOT S102_PRS_I_MT_감지) OR (R102_1_1_M_차종3_LHD AND R102_1_1_M_차종5_MT AND S102_PRS_I_LHD_감지 AND NOT S102_PRS_I_RHD_감지 AND NOT S102_PRS_I_AT_감지 AND S102_PRS_I_MT_감지) OR (R102_1_1_M_차종3_RHD AND R102_1_1_M_차종5_AT AND NOT S102_PRS_I_LHD_감지 AND S102_PRS_I_RHD_감지 AND S102_PRS_I_AT_감지 AND NOT S102_PRS_I_MT_감지) OR (R102_1_1_M_차종3_RHD AND R102_1_1_M_차종5_MT AND NOT S102_PRS_I_LHD_감지 AND S102_PRS_I_RHD_감지 AND NOT S102_PRS_I_AT_감지 AND S102_PRS_I_MT_감지)) AND S102_M_공정_간섭무, PT := T#500MS);
S102_M_공정_사양감지_OK := INST.Q;
(* S102 NONE INT *)
(* Rung L21 *)
S102_M_공정_간섭무 := (R102_1_1_M_I_RB_간섭무_1 OR R102_1_1_M_I_RB_원위치) AND (R102_1_M_I_RB_간섭무_1 OR R102_1_M_I_RB_원위치);
(* R102_1_1 차종 무 *)
(* Rung L24 *)
R102_1_1_M_STN_차종_NONE := NOT R102_1_1_M_STN_차종_ON;

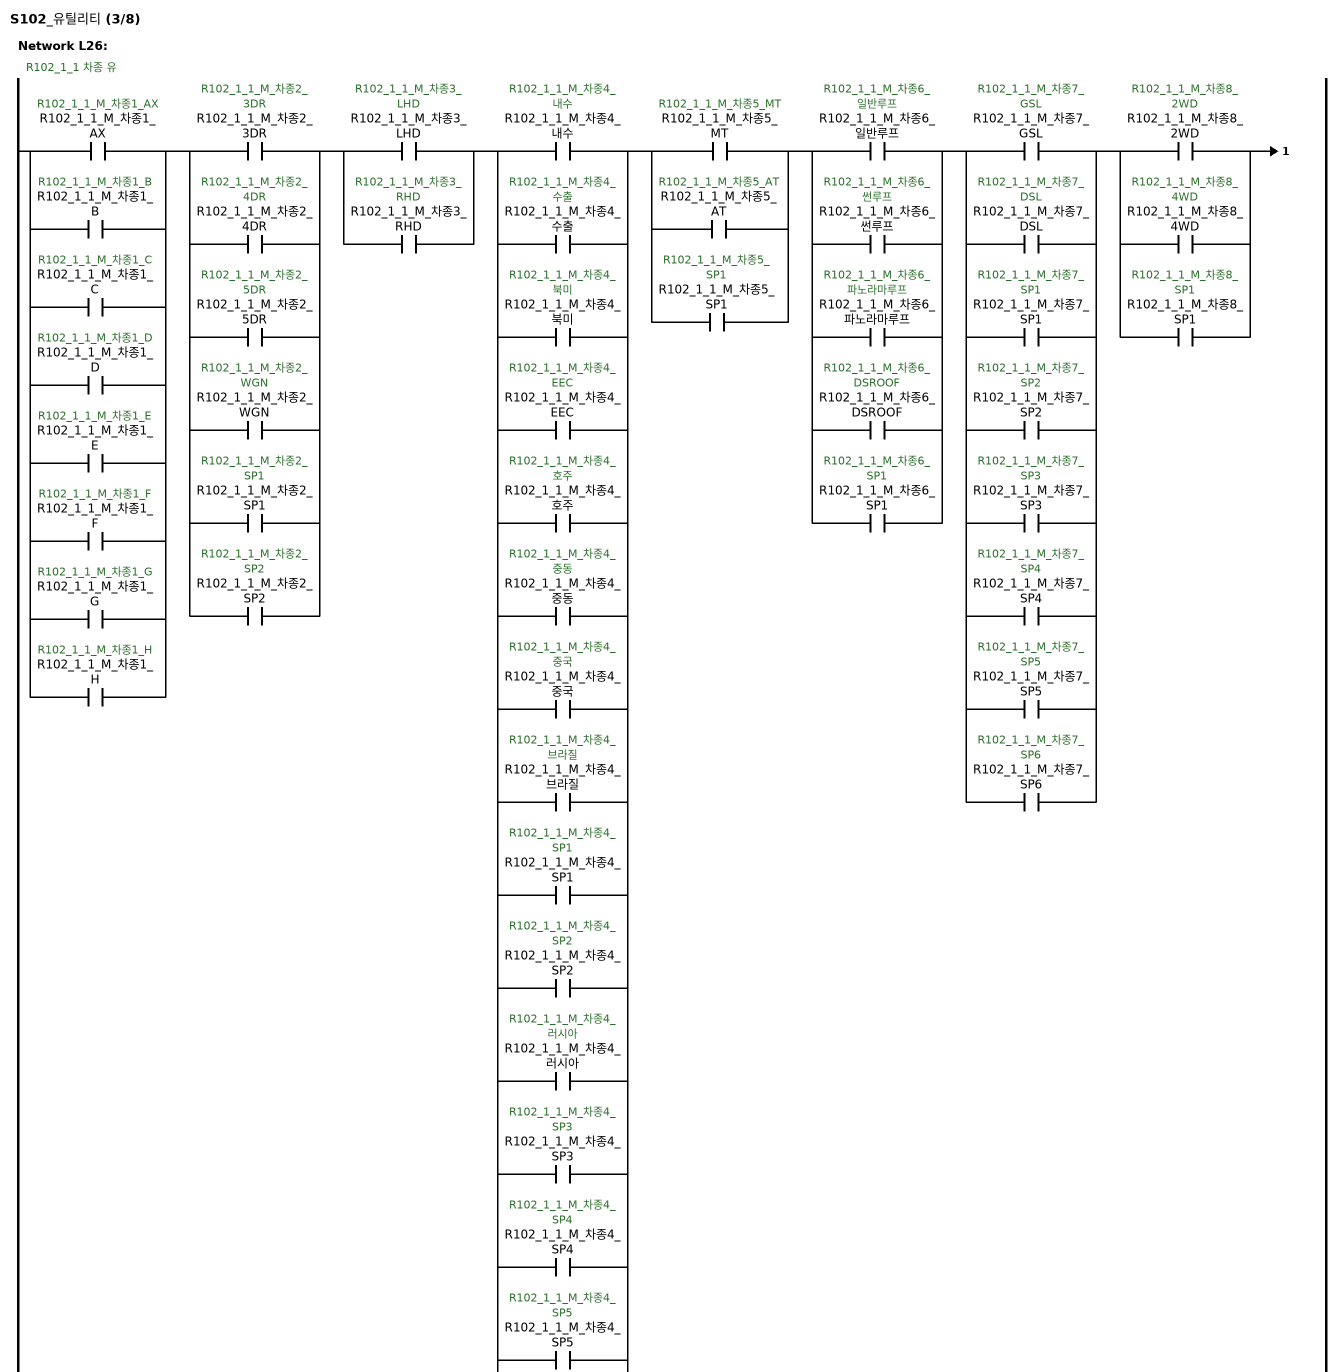

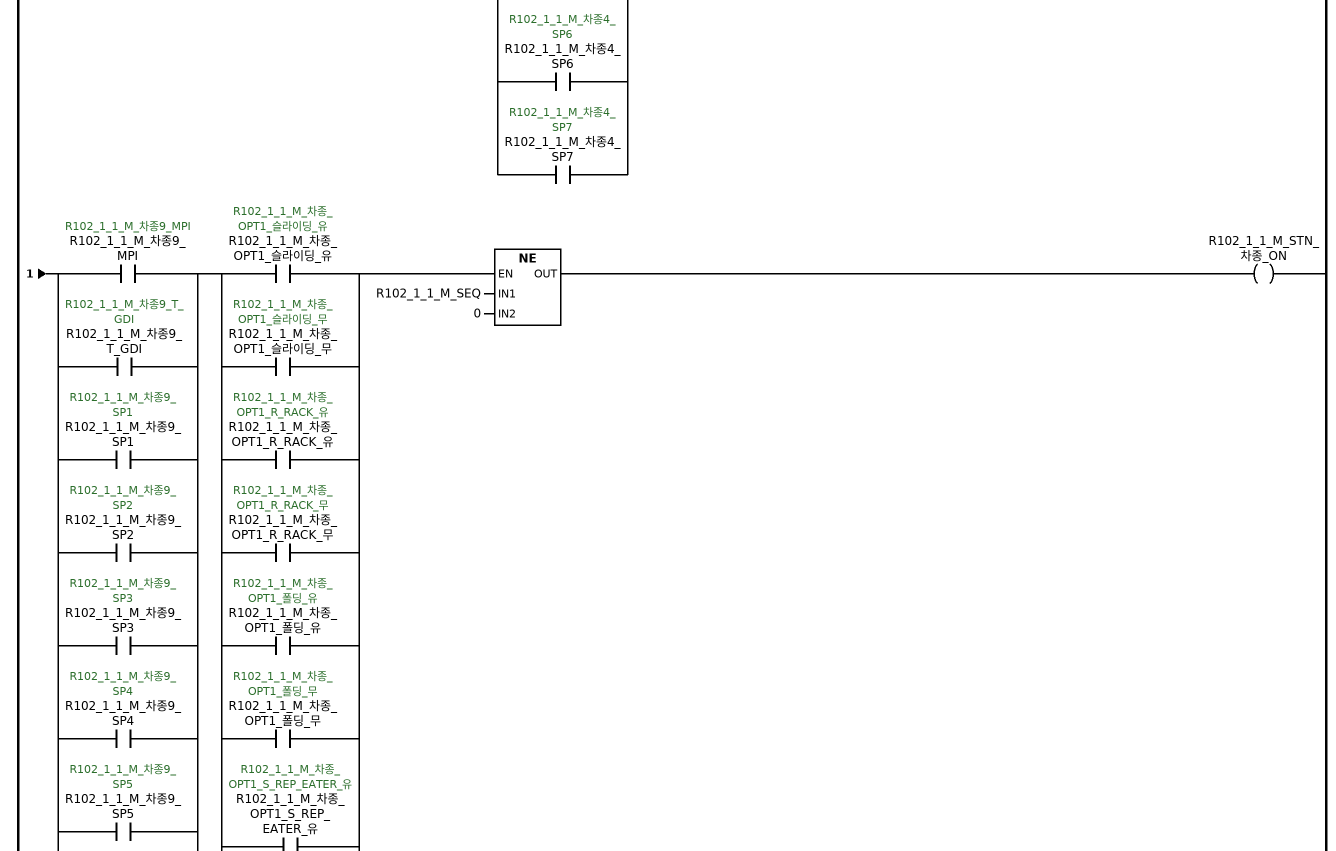

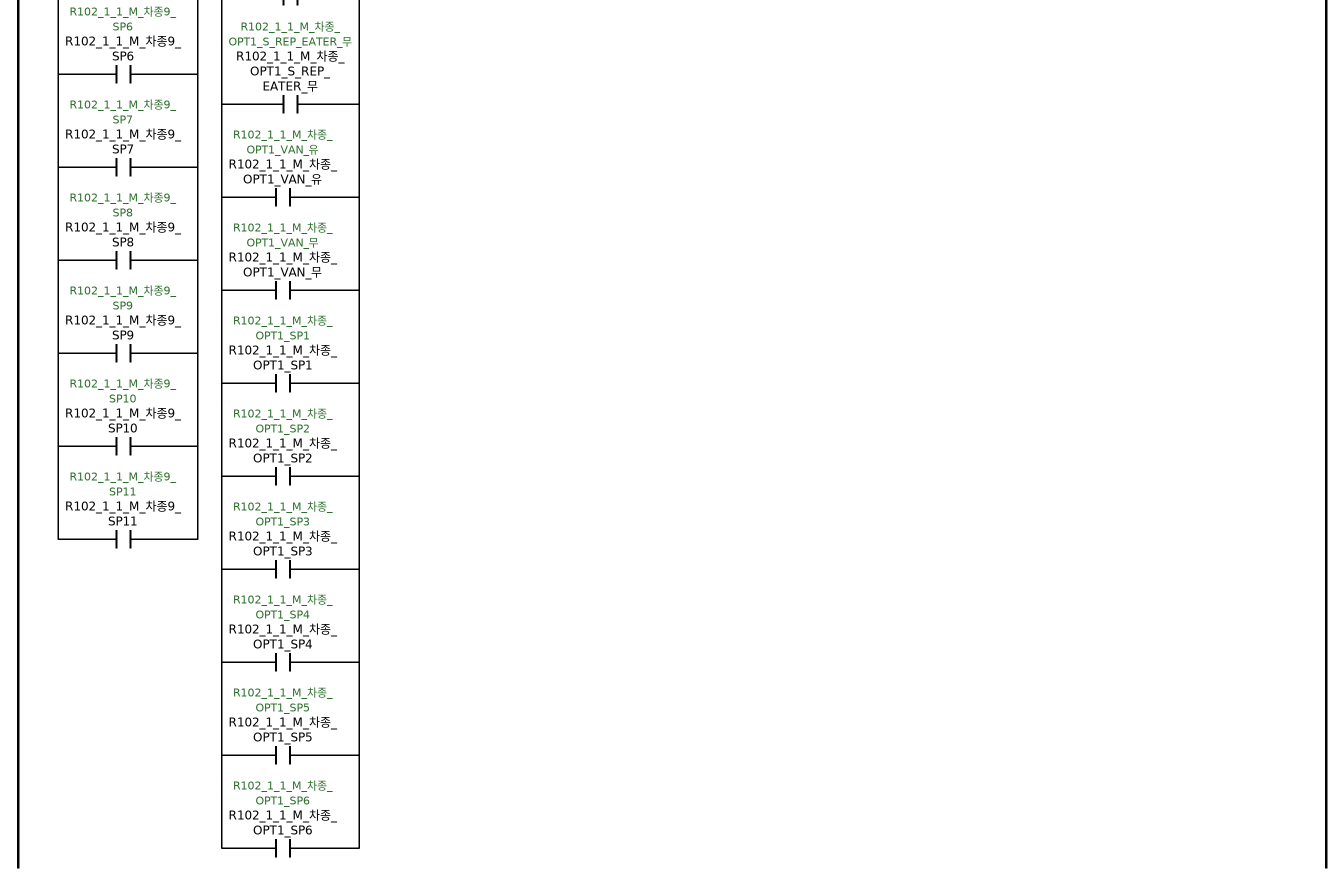
(* R102_1_1 차종 유 *)
(* Rung L26 *)
IF (R102_1_1_M_차종1_AX OR R102_1_1_M_차종1_B OR R102_1_1_M_차종1_C OR R102_1_1_M_차종1_D OR R102_1_1_M_차종1_E OR R102_1_1_M_차종1_F OR R102_1_1_M_차종1_G OR R102_1_1_M_차종1_H) AND (R102_1_1_M_차종2_3DR OR R102_1_1_M_차종2_4DR OR R102_1_1_M_차종2_5DR OR R102_1_1_M_차종2_WGN OR R102_1_1_M_차종2_SP1 OR R102_1_1_M_차종2_SP2) AND (R102_1_1_M_차종3_LHD OR R102_1_1_M_차종3_RHD) AND (R102_1_1_M_차종4_내수 OR R102_1_1_M_차종4_수출 OR R102_1_1_M_차종4_북미 OR R102_1_1_M_차종4_EEC OR R102_1_1_M_차종4_호주 OR R102_1_1_M_차종4_중동 OR R102_1_1_M_차종4_중국 OR R102_1_1_M_차종4_브라질 OR R102_1_1_M_차종4_SP1 OR R102_1_1_M_차종4_SP2 OR R102_1_1_M_차종4_러시아 OR R102_1_1_M_차종4_SP3 OR R102_1_1_M_차종4_SP4 OR R102_1_1_M_차종4_SP5 OR R102_1_1_M_차종4_SP6 OR R102_1_1_M_차종4_SP7) AND (R102_1_1_M_차종5_MT OR R102_1_1_M_차종5_AT OR R102_1_1_M_차종5_SP1) AND (R102_1_1_M_차종6_일반루프 OR R102_1_1_M_차종6_썬루프 OR R102_1_1_M_차종6_파노라마루프 OR R102_1_1_M_차종6_DSROOF OR R102_1_1_M_차종6_SP1) AND (R102_1_1_M_차종7_GSL OR R102_1_1_M_차종7_DSL OR R102_1_1_M_차종7_SP1 OR R102_1_1_M_차종7_SP2 OR R102_1_1_M_차종7_SP3 OR R102_1_1_M_차종7_SP4 OR R102_1_1_M_차종7_SP5 OR R102_1_1_M_차종7_SP6) AND (R102_1_1_M_차종8_2WD OR R102_1_1_M_차종8_4WD OR R102_1_1_M_차종8_SP1) AND (R102_1_1_M_차종9_MPI OR R102_1_1_M_차종9_T_GDI OR R102_1_1_M_차종9_SP1 OR R102_1_1_M_차종9_SP2 OR R102_1_1_M_차종9_SP3 OR R102_1_1_M_차종9_SP4 OR R102_1_1_M_차종9_SP5 OR R102_1_1_M_차종9_SP6 OR R102_1_1_M_차종9_SP7 OR R102_1_1_M_차종9_SP8 OR R102_1_1_M_차종9_SP9 OR R102_1_1_M_차종9_SP10 OR R102_1_1_M_차종9_SP11) AND (R102_1_1_M_차종_OPT1_슬라이딩_유 OR R102_1_1_M_차종_OPT1_슬라이딩_무 OR R102_1_1_M_차종_OPT1_R_RACK_유 OR R102_1_1_M_차종_OPT1_R_RACK_무 OR R102_1_1_M_차종_OPT1_폴딩_유 OR R102_1_1_M_차종_OPT1_폴딩_무 OR R102_1_1_M_차종_OPT1_S_REP_EATER_유 OR R102_1_1_M_차종_OPT1_S_REP_EATER_무 OR R102_1_1_M_차종_OPT1_VAN_유 OR R102_1_1_M_차종_OPT1_VAN_무 OR R102_1_1_M_차종_OPT1_SP1 OR R102_1_1_M_차종_OPT1_SP2 OR R102_1_1_M_차종_OPT1_SP3 OR R102_1_1_M_차종_OPT1_SP4 OR R102_1_1_M_차종_OPT1_SP5 OR R102_1_1_M_차종_OPT1_SP6) THEN
    _t1 := R102_1_1_M_SEQ <> 0;
END_IF;
R102_1_1_M_STN_차종_ON := _t1;

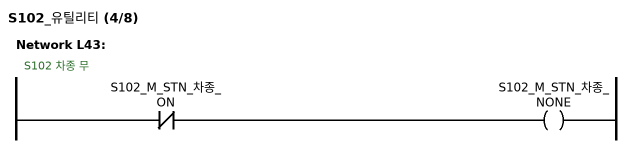
(* S102 차종 무 *)
(* Rung L43 *)
S102_M_STN_차종_NONE := NOT S102_M_STN_차종_ON;

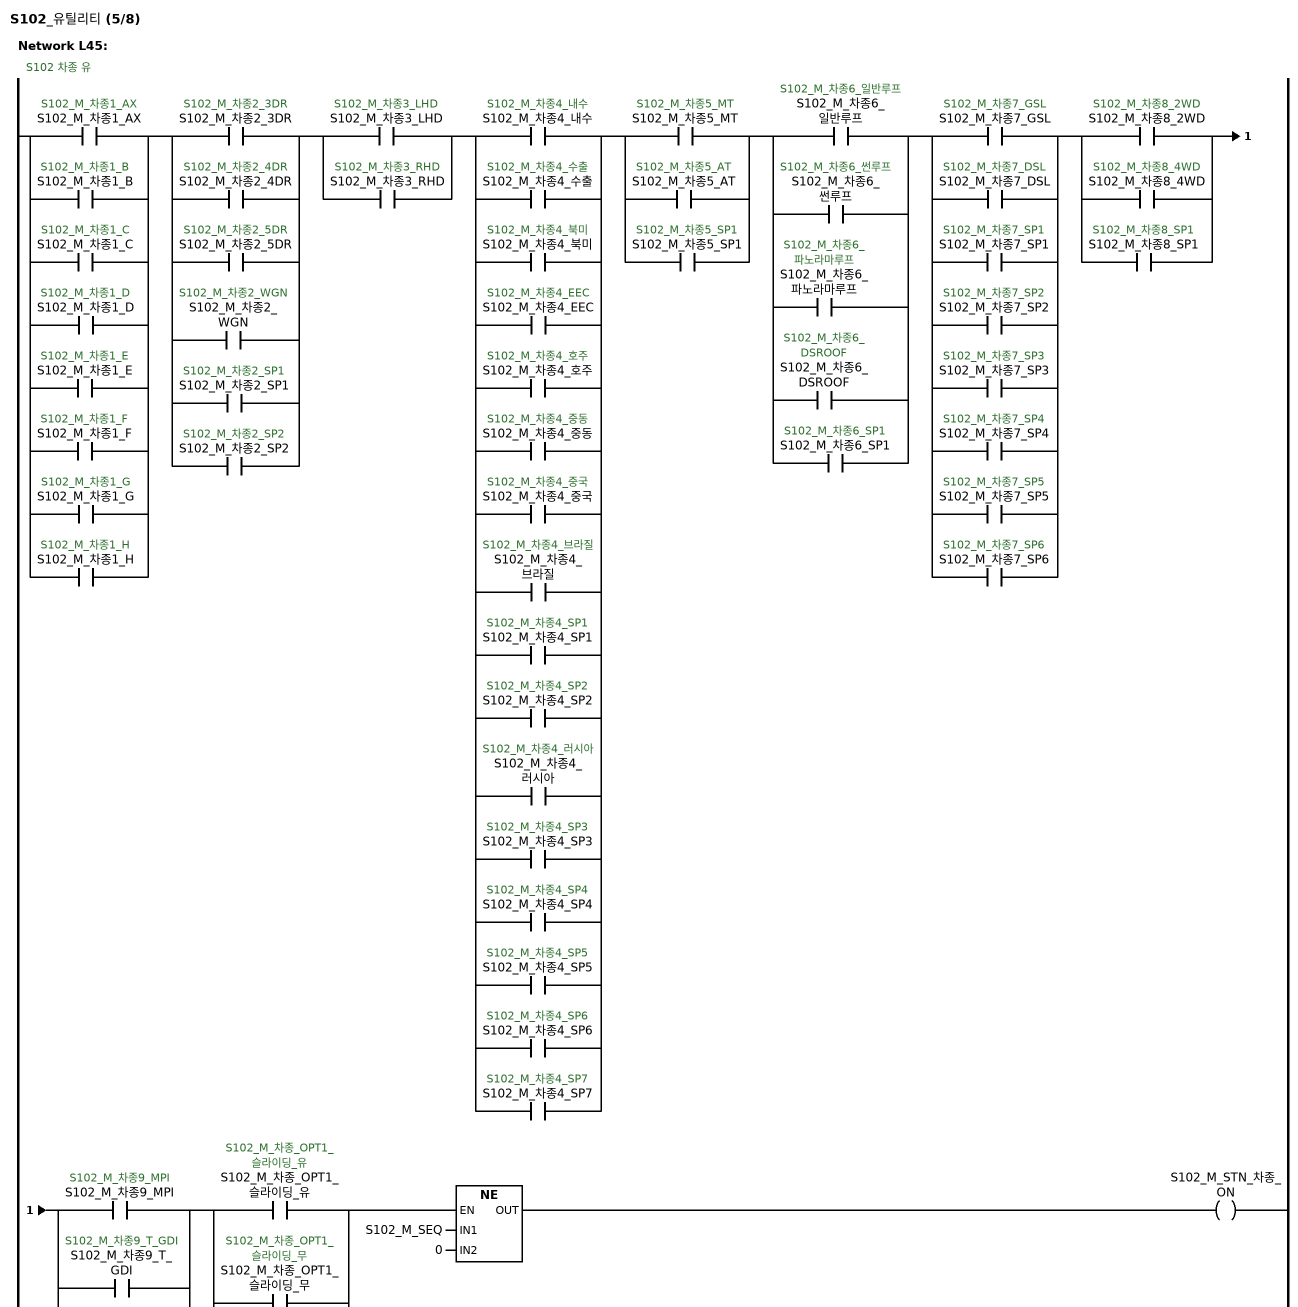

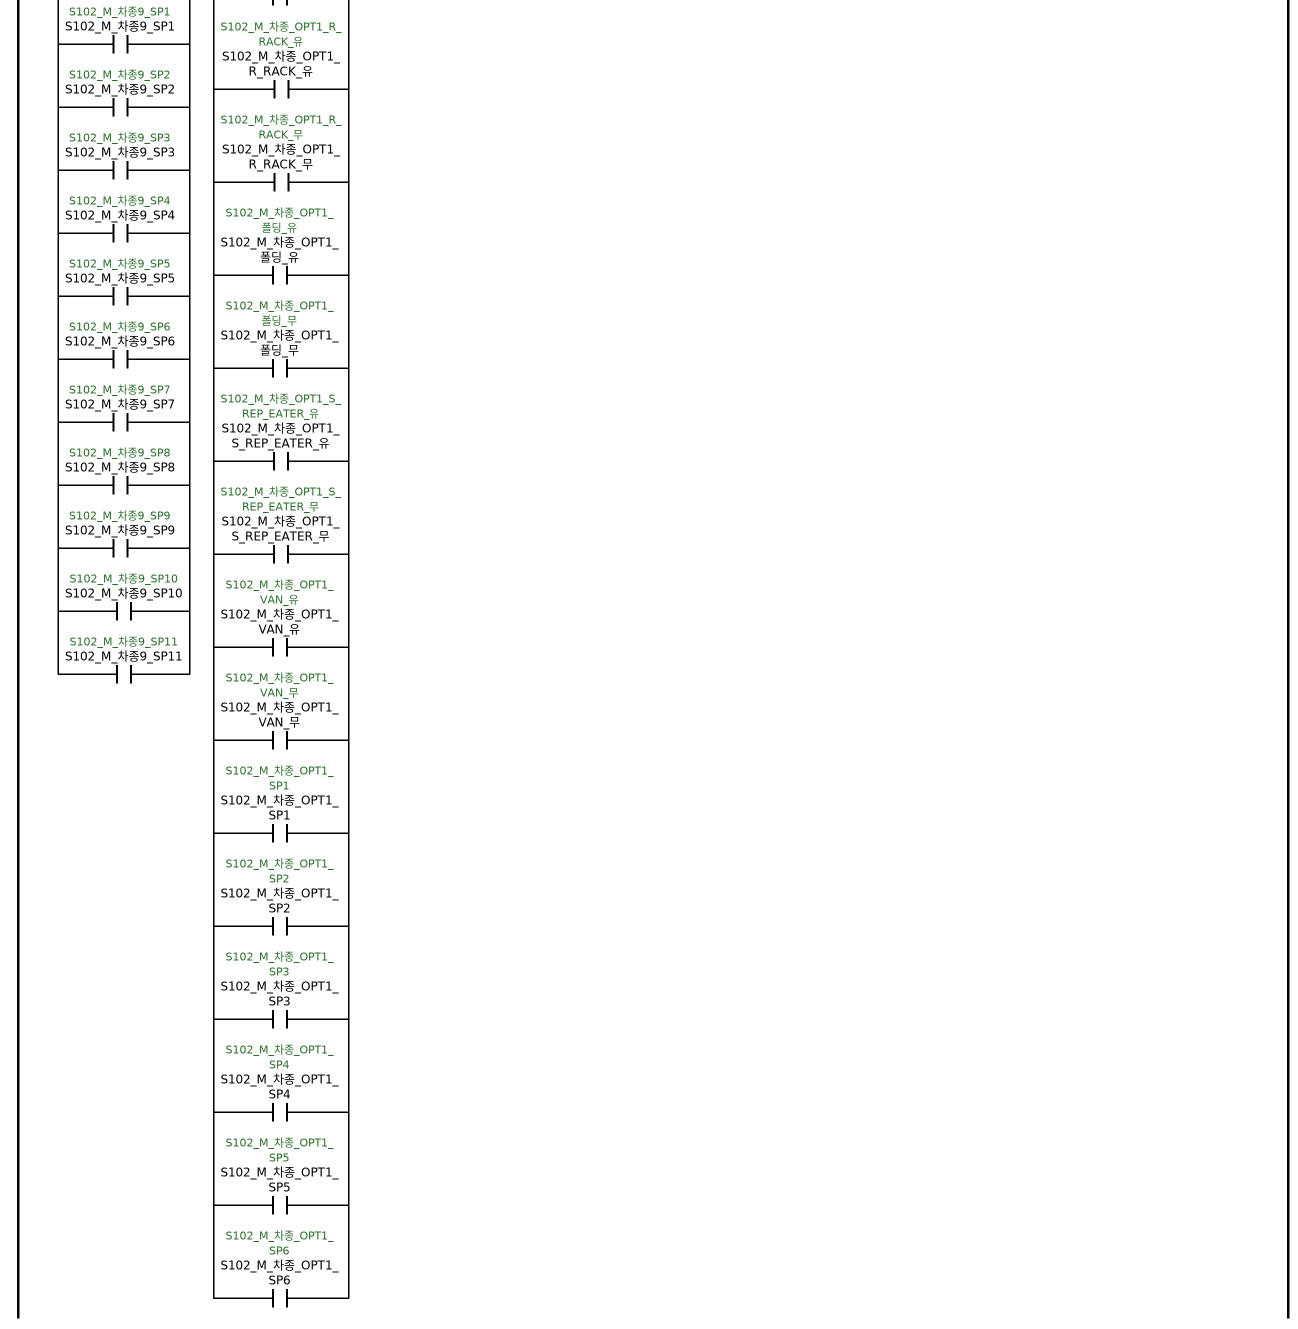
(* S102 차종 유 *)
(* Rung L45 *)
IF (S102_M_차종1_AX OR S102_M_차종1_B OR S102_M_차종1_C OR S102_M_차종1_D OR S102_M_차종1_E OR S102_M_차종1_F OR S102_M_차종1_G OR S102_M_차종1_H) AND (S102_M_차종2_3DR OR S102_M_차종2_4DR OR S102_M_차종2_5DR OR S102_M_차종2_WGN OR S102_M_차종2_SP1 OR S102_M_차종2_SP2) AND (S102_M_차종3_LHD OR S102_M_차종3_RHD) AND (S102_M_차종4_내수 OR S102_M_차종4_수출 OR S102_M_차종4_북미 OR S102_M_차종4_EEC OR S102_M_차종4_호주 OR S102_M_차종4_중동 OR S102_M_차종4_중국 OR S102_M_차종4_브라질 OR S102_M_차종4_SP1 OR S102_M_차종4_SP2 OR S102_M_차종4_러시아 OR S102_M_차종4_SP3 OR S102_M_차종4_SP4 OR S102_M_차종4_SP5 OR S102_M_차종4_SP6 OR S102_M_차종4_SP7) AND (S102_M_차종5_MT OR S102_M_차종5_AT OR S102_M_차종5_SP1) AND (S102_M_차종6_일반루프 OR S102_M_차종6_썬루프 OR S102_M_차종6_파노라마루프 OR S102_M_차종6_DSROOF OR S102_M_차종6_SP1) AND (S102_M_차종7_GSL OR S102_M_차종7_DSL OR S102_M_차종7_SP1 OR S102_M_차종7_SP2 OR S102_M_차종7_SP3 OR S102_M_차종7_SP4 OR S102_M_차종7_SP5 OR S102_M_차종7_SP6) AND (S102_M_차종8_2WD OR S102_M_차종8_4WD OR S102_M_차종8_SP1) AND (S102_M_차종9_MPI OR S102_M_차종9_T_GDI OR S102_M_차종9_SP1 OR S102_M_차종9_SP2 OR S102_M_차종9_SP3 OR S102_M_차종9_SP4 OR S102_M_차종9_SP5 OR S102_M_차종9_SP6 OR S102_M_차종9_SP7 OR S102_M_차종9_SP8 OR S102_M_차종9_SP9 OR S102_M_차종9_SP10 OR S102_M_차종9_SP11) AND (S102_M_차종_OPT1_슬라이딩_유 OR S102_M_차종_OPT1_슬라이딩_무 OR S102_M_차종_OPT1_R_RACK_유 OR S102_M_차종_OPT1_R_RACK_무 OR S102_M_차종_OPT1_폴딩_유 OR S102_M_차종_OPT1_폴딩_무 OR S102_M_차종_OPT1_S_REP_EATER_유 OR S102_M_차종_OPT1_S_REP_EATER_무 OR S102_M_차종_OPT1_VAN_유 OR S102_M_차종_OPT1_VAN_무 OR S102_M_차종_OPT1_SP1 OR S102_M_차종_OPT1_SP2 OR S102_M_차종_OPT1_SP3 OR S102_M_차종_OPT1_SP4 OR S102_M_차종_OPT1_SP5 OR S102_M_차종_OPT1_SP6) THEN
    _t2 := S102_M_SEQ <> 0;
END_IF;
S102_M_STN_차종_ON := _t2;

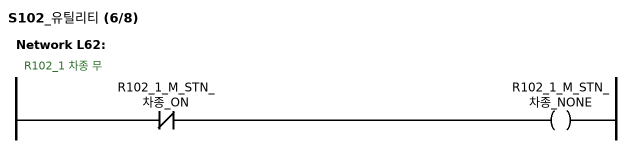
(* R102_1 차종 무 *)
(* Rung L62 *)
R102_1_M_STN_차종_NONE := NOT R102_1_M_STN_차종_ON;

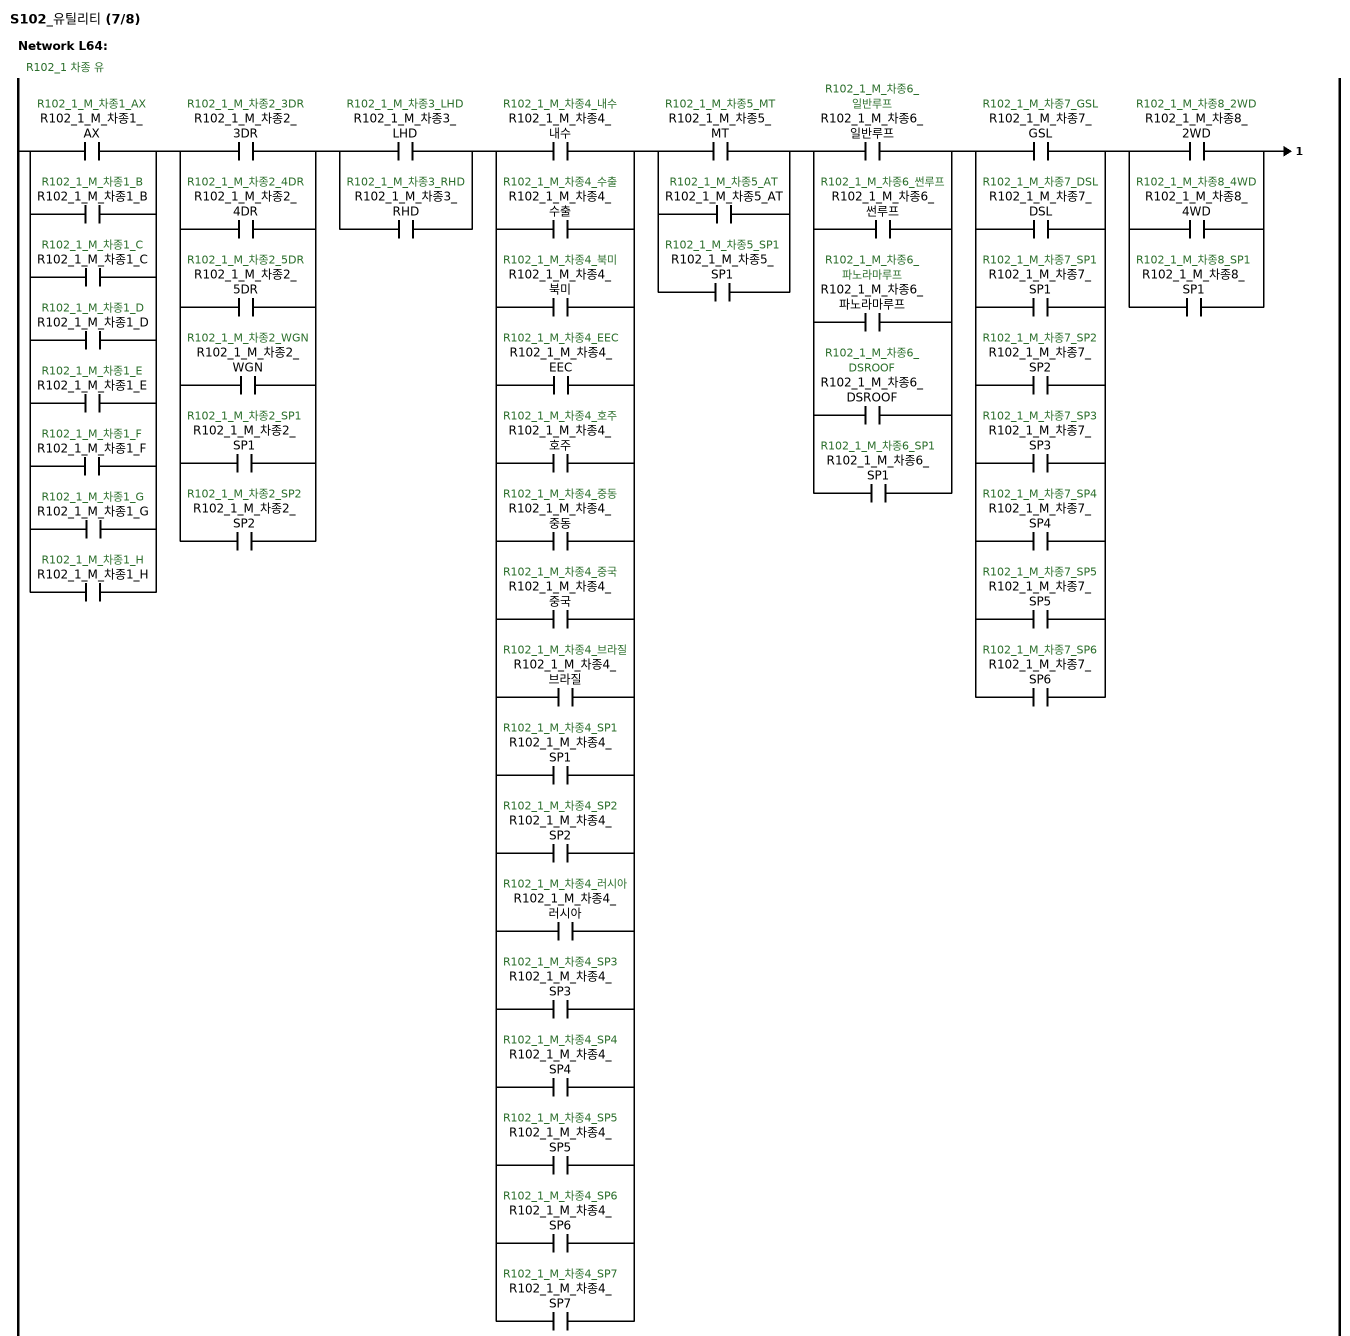

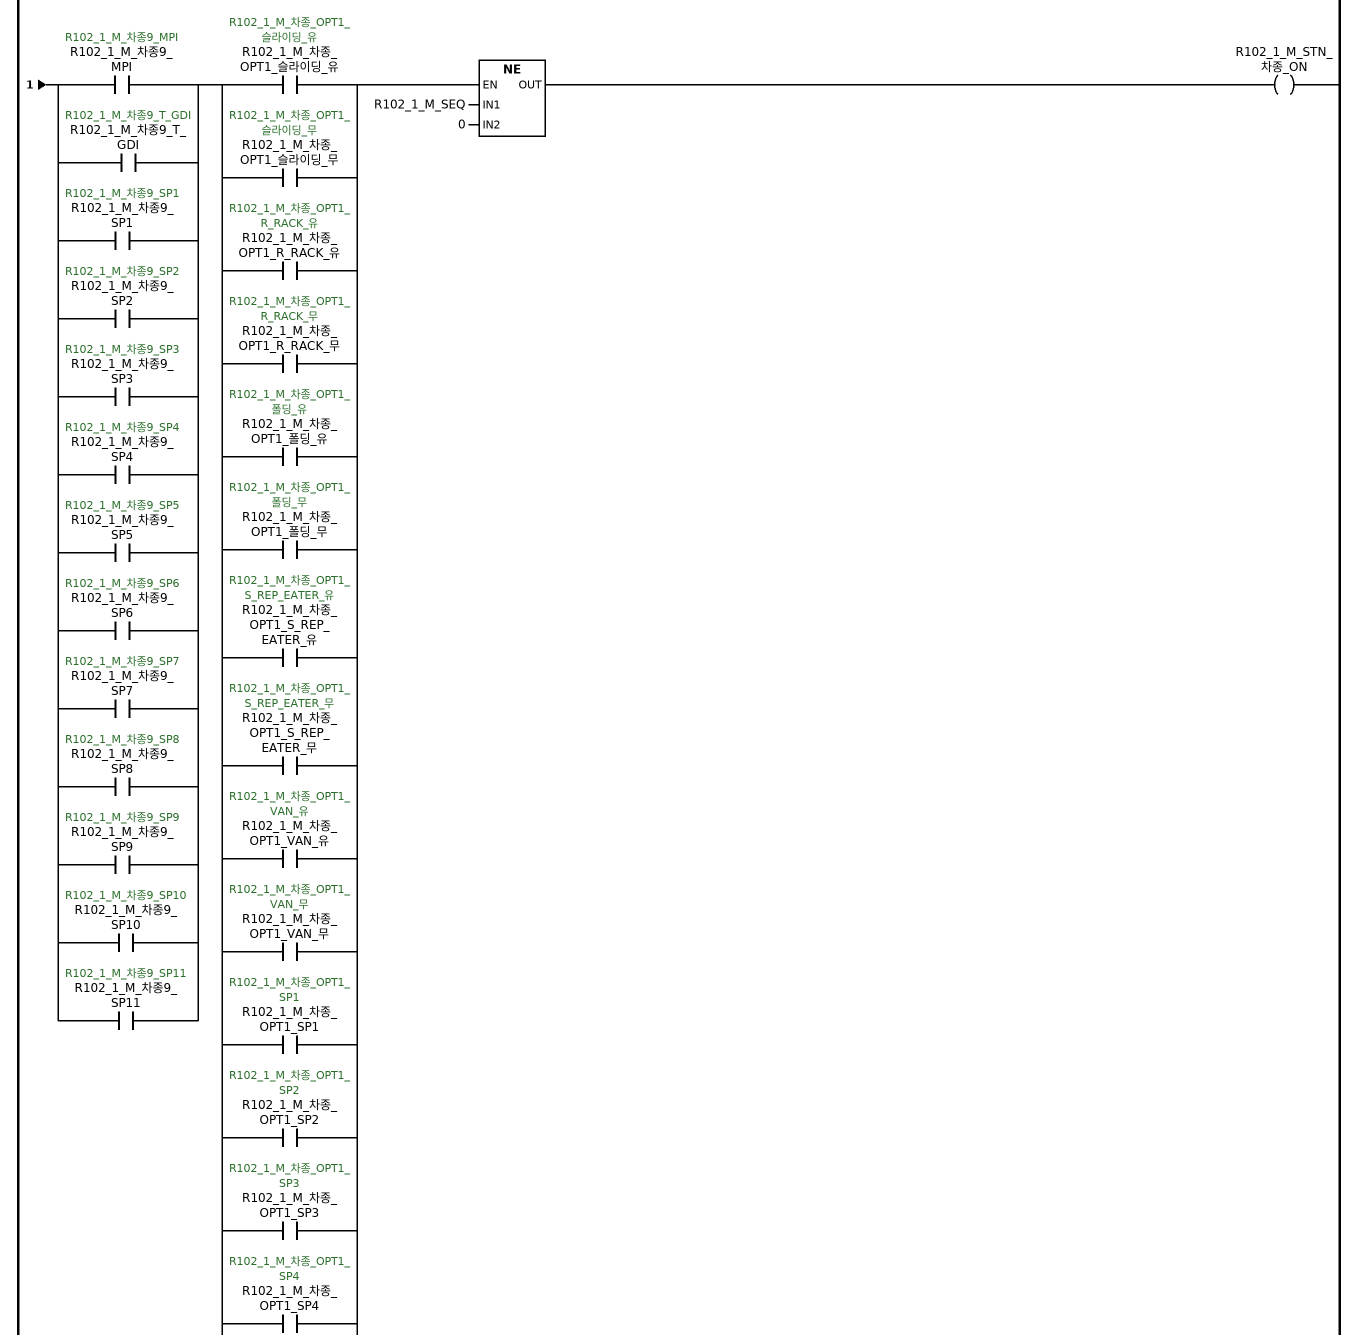

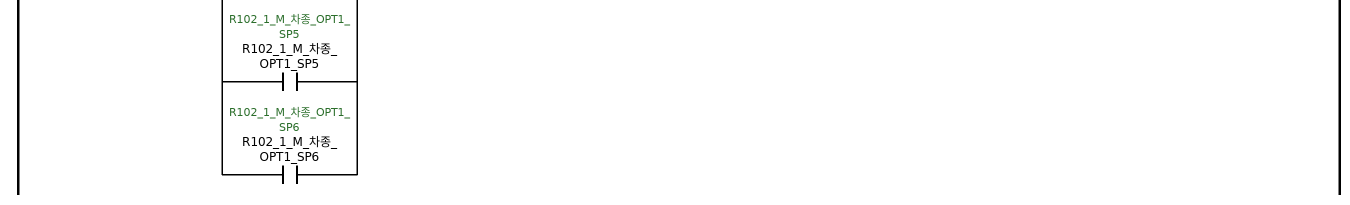
(* R102_1 차종 유 *)
(* Rung L64 *)
IF (R102_1_M_차종1_AX OR R102_1_M_차종1_B OR R102_1_M_차종1_C OR R102_1_M_차종1_D OR R102_1_M_차종1_E OR R102_1_M_차종1_F OR R102_1_M_차종1_G OR R102_1_M_차종1_H) AND (R102_1_M_차종2_3DR OR R102_1_M_차종2_4DR OR R102_1_M_차종2_5DR OR R102_1_M_차종2_WGN OR R102_1_M_차종2_SP1 OR R102_1_M_차종2_SP2) AND (R102_1_M_차종3_LHD OR R102_1_M_차종3_RHD) AND (R102_1_M_차종4_내수 OR R102_1_M_차종4_수출 OR R102_1_M_차종4_북미 OR R102_1_M_차종4_EEC OR R102_1_M_차종4_호주 OR R102_1_M_차종4_중동 OR R102_1_M_차종4_중국 OR R102_1_M_차종4_브라질 OR R102_1_M_차종4_SP1 OR R102_1_M_차종4_SP2 OR R102_1_M_차종4_러시아 OR R102_1_M_차종4_SP3 OR R102_1_M_차종4_SP4 OR R102_1_M_차종4_SP5 OR R102_1_M_차종4_SP6 OR R102_1_M_차종4_SP7) AND (R102_1_M_차종5_MT OR R102_1_M_차종5_AT OR R102_1_M_차종5_SP1) AND (R102_1_M_차종6_일반루프 OR R102_1_M_차종6_썬루프 OR R102_1_M_차종6_파노라마루프 OR R102_1_M_차종6_DSROOF OR R102_1_M_차종6_SP1) AND (R102_1_M_차종7_GSL OR R102_1_M_차종7_DSL OR R102_1_M_차종7_SP1 OR R102_1_M_차종7_SP2 OR R102_1_M_차종7_SP3 OR R102_1_M_차종7_SP4 OR R102_1_M_차종7_SP5 OR R102_1_M_차종7_SP6) AND (R102_1_M_차종8_2WD OR R102_1_M_차종8_4WD OR R102_1_M_차종8_SP1) AND (R102_1_M_차종9_MPI OR R102_1_M_차종9_T_GDI OR R102_1_M_차종9_SP1 OR R102_1_M_차종9_SP2 OR R102_1_M_차종9_SP3 OR R102_1_M_차종9_SP4 OR R102_1_M_차종9_SP5 OR R102_1_M_차종9_SP6 OR R102_1_M_차종9_SP7 OR R102_1_M_차종9_SP8 OR R102_1_M_차종9_SP9 OR R102_1_M_차종9_SP10 OR R102_1_M_차종9_SP11) AND (R102_1_M_차종_OPT1_슬라이딩_유 OR R102_1_M_차종_OPT1_슬라이딩_무 OR R102_1_M_차종_OPT1_R_RACK_유 OR R102_1_M_차종_OPT1_R_RACK_무 OR R102_1_M_차종_OPT1_폴딩_유 OR R102_1_M_차종_OPT1_폴딩_무 OR R102_1_M_차종_OPT1_S_REP_EATER_유 OR R102_1_M_차종_OPT1_S_REP_EATER_무 OR R102_1_M_차종_OPT1_VAN_유 OR R102_1_M_차종_OPT1_VAN_무 OR R102_1_M_차종_OPT1_SP1 OR R102_1_M_차종_OPT1_SP2 OR R102_1_M_차종_OPT1_SP3 OR R102_1_M_차종_OPT1_SP4 OR R102_1_M_차종_OPT1_SP5 OR R102_1_M_차종_OPT1_SP6) THEN
    _t3 := R102_1_M_SEQ <> 0;
END_IF;
R102_1_M_STN_차종_ON := _t3;

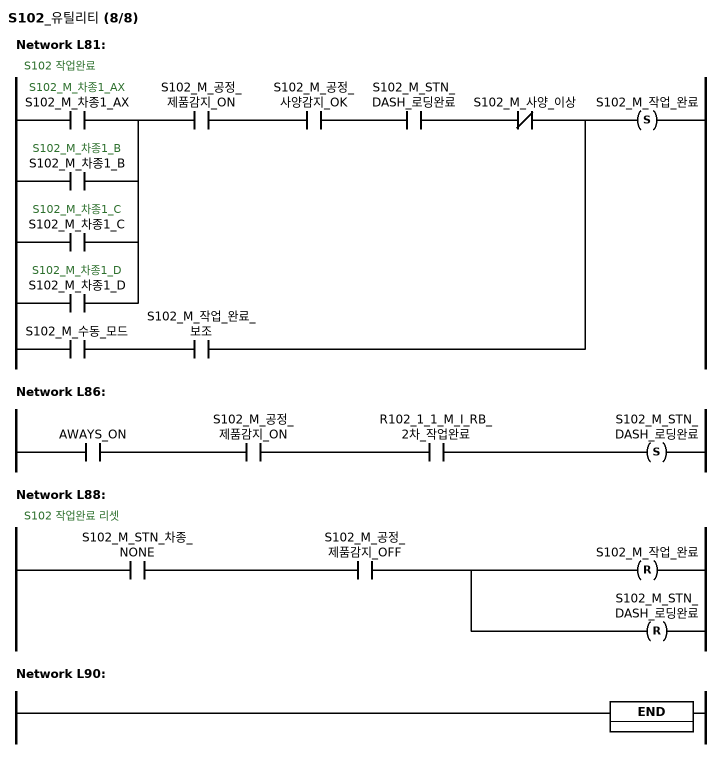
(* S102 작업완료 *)
(* Rung L81 *)
IF ((S102_M_차종1_AX OR S102_M_차종1_B OR S102_M_차종1_C OR S102_M_차종1_D) AND S102_M_공정_제품감지_ON AND S102_M_공정_사양감지_OK AND S102_M_STN_DASH_로딩완료 AND NOT S102_M_사양_이상) OR (S102_M_수동_모드 AND S102_M_작업_완료_보조) THEN
    S102_M_작업_완료 := TRUE;
END_IF;
(* Rung L86 *)
IF AWAYS_ON AND S102_M_공정_제품감지_ON AND R102_1_1_M_I_RB_2차_작업완료 THEN S102_M_STN_DASH_로딩완료 := TRUE; END_IF;
(* S102 작업완료 리셋 *)
(* Rung L88 *)
IF S102_M_STN_차종_NONE AND S102_M_공정_제품감지_OFF THEN
    S102_M_작업_완료 := FALSE;
    S102_M_STN_DASH_로딩완료 := FALSE;
END_IF;
(* Rung L90 *)
END();
END_PROGRAM

PROGRAM S102_DASH_랙방 (* task: 스캔 프로그램 *)
VAR_EXTERNAL
    AWAYS_ON : BOOL; (* AT %MW3.1 *)
    DASH_RACK1_I_막장감지 : BOOL; (* AT %MW87300.2 *)
    DASH_RACK1_I_종발이감지1 : BOOL; (* AT %MW87300.0 *)
    DASH_RACK1_I_종발이감지2 : BOOL; (* AT %MW87300.1 *)
    DASH_RACK2_I_막장감지 : BOOL; (* AT %MW87300.10 *)
    DASH_RACK2_I_종발이감지1 : BOOL; (* AT %MW87300.8 *)
    DASH_RACK2_I_종발이감지2 : BOOL; (* AT %MW87300.9 *)
    DASH_RACK3_I_막장감지 : BOOL; (* AT %MW87301.2 *)
    DASH_RACK3_I_종발이감지1 : BOOL; (* AT %MW87301.0 *)
    DASH_RACK3_I_종발이감지2 : BOOL; (* AT %MW87301.1 *)
    DASH_RACK4_I_막장감지 : BOOL; (* AT %MW87301.10 *)
    DASH_RACK4_I_종발이감지1 : BOOL; (* AT %MW87301.8 *)
    DASH_RACK4_I_종발이감지2 : BOOL; (* AT %MW87301.9 *)
    OTR_RACK1_I_막장감지 : BOOL; (* AT %MW87020.2 *)
    OTR_RACK1_I_종발이감지1 : BOOL; (* AT %MW87020.0 *)
    OTR_RACK1_I_종발이감지2 : BOOL; (* AT %MW87020.1 *)
    OTR_RACK2_I_막장감지 : BOOL; (* AT %MW87020.10 *)
    OTR_RACK2_I_종발이감지1 : BOOL; (* AT %MW87020.8 *)
    OTR_RACK2_I_종발이감지2 : BOOL; (* AT %MW87020.9 *)
    R101_1_M_RB_PROG_NO : WORD; (* AT %MW20074 *)
    R102_1_1_M_RB_PROG_NO : WORD; (* AT %MW20094 *)
    S101_LH_M_APRON_PLT1_FAULT : BOOL; (* AT %MW1200.6 *)
    S101_LH_M_APRON_PLT1_MATCH_OK : BOOL; (* AT %MW1200.5 *)
    S101_LH_M_APRON_PLT1_PLT_NONE : BOOL; (* AT %MW1200.2 *)
    S101_LH_M_APRON_PLT1_PLT_ON : BOOL; (* AT %MW1200.1 *)
    S101_LH_M_APRON_PLT1_PROG_OK : BOOL; (* AT %MW1200.0 *)
    S101_LH_M_APRON_PLT1_로딩완료 : BOOL; (* AT %MW1200.10 *)
    S101_LH_M_APRON_PLT1_제품수량 : WORD; (* AT %MW1224 *)
    S101_LH_M_APRON_PLT1_차종유 : BOOL; (* AT %MW1200.8 *)
    S101_LH_M_APRON_PLT1_차종코드 : WORD; (* AT %MW1216 *)
    S101_LH_M_APRON_PLT1_파트무 : BOOL; (* AT %MW1200.4 *)
    S101_LH_M_APRON_PLT1_파트유 : BOOL; (* AT %MW1200.3 *)
    S101_LH_M_APRON_PLT2_FAULT : BOOL; (* AT %MW1201.6 *)
    S101_LH_M_APRON_PLT2_MATCH_OK : BOOL; (* AT %MW1201.5 *)
    S101_LH_M_APRON_PLT2_PLT_NONE : BOOL; (* AT %MW1201.2 *)
    S101_LH_M_APRON_PLT2_PLT_ON : BOOL; (* AT %MW1201.1 *)
    S101_LH_M_APRON_PLT2_PROG_OK : BOOL; (* AT %MW1201.0 *)
    S101_LH_M_APRON_PLT2_로딩완료 : BOOL; (* AT %MW1201.10 *)
    S101_LH_M_APRON_PLT2_제품수량 : WORD; (* AT %MW1225 *)
    S101_LH_M_APRON_PLT2_차종유 : BOOL; (* AT %MW1201.8 *)
    S101_LH_M_APRON_PLT2_차종코드 : WORD; (* AT %MW1217 *)
    S101_LH_M_APRON_PLT2_파트무 : BOOL; (* AT %MW1201.4 *)
    S101_LH_M_APRON_PLT2_파트유 : BOOL; (* AT %MW1201.3 *)
    S101_RH_M_APRON_PLT1_FAULT : BOOL; (* AT %MW1250.6 *)
    S101_RH_M_APRON_PLT1_MATCH_OK : BOOL; (* AT %MW1250.5 *)
    S101_RH_M_APRON_PLT1_PLT_NONE : BOOL; (* AT %MW1250.2 *)
    S101_RH_M_APRON_PLT1_PLT_ON : BOOL; (* AT %MW1250.1 *)
    S101_RH_M_APRON_PLT1_PROG_OK : BOOL; (* AT %MW1250.0 *)
    S101_RH_M_APRON_PLT1_로딩완료 : BOOL; (* AT %MW1250.10 *)
    S101_RH_M_APRON_PLT1_제품수량 : WORD; (* AT %MW1274 *)
    S101_RH_M_APRON_PLT1_차종유 : BOOL; (* AT %MW1250.8 *)
    S101_RH_M_APRON_PLT1_차종코드 : WORD; (* AT %MW1266 *)
    S101_RH_M_APRON_PLT1_파트무 : BOOL;
    S101_RH_M_APRON_PLT1_파트유 : BOOL; (* AT %MW1250.3 *)
    S101_RH_M_APRON_PLT2_FAULT : BOOL; (* AT %MW1251.6 *)
    S101_RH_M_APRON_PLT2_MATCH_OK : BOOL; (* AT %MW1251.5 *)
    S101_RH_M_APRON_PLT2_PLT_NONE : BOOL; (* AT %MW1251.2 *)
    S101_RH_M_APRON_PLT2_PLT_ON : BOOL; (* AT %MW1251.1 *)
    S101_RH_M_APRON_PLT2_PROG_OK : BOOL; (* AT %MW1251.0 *)
    S101_RH_M_APRON_PLT2_로딩완료 : BOOL; (* AT %MW1251.10 *)
    S101_RH_M_APRON_PLT2_제품수량 : WORD; (* AT %MW1275 *)
    S101_RH_M_APRON_PLT2_차종유 : BOOL; (* AT %MW1251.8 *)
    S101_RH_M_APRON_PLT2_차종코드 : WORD; (* AT %MW1267 *)
    S101_RH_M_APRON_PLT2_파트무 : BOOL; (* AT %MW1251.4 *)
    S101_RH_M_APRON_PLT2_파트유 : BOOL; (* AT %MW1251.3 *)
    S102_M_DASH_PLT1_FAULT : BOOL; (* AT %MW1700.6 *)
    S102_M_DASH_PLT1_MATCH_OK : BOOL; (* AT %MW1700.5 *)
    S102_M_DASH_PLT1_PLT_NONE : BOOL; (* AT %MW1700.2 *)
    S102_M_DASH_PLT1_PLT_ON : BOOL; (* AT %MW1700.1 *)
    S102_M_DASH_PLT1_PROG_OK : BOOL; (* AT %MW1700.0 *)
    S102_M_DASH_PLT1_로딩완료 : BOOL; (* AT %MW1700.10 *)
    S102_M_DASH_PLT1_제품수량 : WORD; (* AT %MW1724 *)
    S102_M_DASH_PLT1_차종유 : BOOL; (* AT %MW1700.8 *)
    S102_M_DASH_PLT1_차종코드 : WORD; (* AT %MW1716 *)
    S102_M_DASH_PLT1_파트무 : BOOL; (* AT %MW1700.4 *)
    S102_M_DASH_PLT1_파트유 : BOOL; (* AT %MW1700.3 *)
    S102_M_DASH_PLT2_FAULT : BOOL; (* AT %MW1701.6 *)
    S102_M_DASH_PLT2_MATCH_OK : BOOL; (* AT %MW1701.5 *)
    S102_M_DASH_PLT2_PLT_NONE : BOOL; (* AT %MW1701.2 *)
    S102_M_DASH_PLT2_PLT_ON : BOOL; (* AT %MW1701.1 *)
    S102_M_DASH_PLT2_PROG_OK : BOOL; (* AT %MW1701.0 *)
    S102_M_DASH_PLT2_로딩완료 : BOOL; (* AT %MW1701.10 *)
    S102_M_DASH_PLT2_제품수량 : WORD; (* AT %MW1725 *)
    S102_M_DASH_PLT2_차종유 : BOOL; (* AT %MW1701.8 *)
    S102_M_DASH_PLT2_차종코드 : WORD; (* AT %MW1717 *)
    S102_M_DASH_PLT2_파트무 : BOOL; (* AT %MW1701.4 *)
    S102_M_DASH_PLT2_파트유 : BOOL; (* AT %MW1701.3 *)
    S102_M_DASH_PLT3_FAULT : BOOL; (* AT %MW1702.6 *)
    S102_M_DASH_PLT3_MATCH_OK : BOOL; (* AT %MW1702.5 *)
    S102_M_DASH_PLT3_PLT_NONE : BOOL; (* AT %MW1702.2 *)
    S102_M_DASH_PLT3_PLT_ON : BOOL; (* AT %MW1702.1 *)
    S102_M_DASH_PLT3_PROG_OK : BOOL; (* AT %MW1702.0 *)
    S102_M_DASH_PLT3_로딩완료 : BOOL; (* AT %MW1702.10 *)
    S102_M_DASH_PLT3_제품수량 : WORD; (* AT %MW1726 *)
    S102_M_DASH_PLT3_차종유 : BOOL; (* AT %MW1702.8 *)
    S102_M_DASH_PLT3_차종코드 : WORD; (* AT %MW1718 *)
    S102_M_DASH_PLT3_파트무 : BOOL; (* AT %MW1702.4 *)
    S102_M_DASH_PLT3_파트유 : BOOL; (* AT %MW1702.3 *)
    S102_M_DASH_PLT4_FAULT : BOOL; (* AT %MW1703.6 *)
    S102_M_DASH_PLT4_MATCH_OK : BOOL; (* AT %MW1703.5 *)
    S102_M_DASH_PLT4_PLT_NONE : BOOL; (* AT %MW1703.2 *)
    S102_M_DASH_PLT4_PLT_ON : BOOL; (* AT %MW1703.1 *)
    S102_M_DASH_PLT4_PROG_OK : BOOL; (* AT %MW1703.0 *)
    S102_M_DASH_PLT4_로딩완료 : BOOL; (* AT %MW1703.10 *)
    S102_M_DASH_PLT4_제품수량 : WORD; (* AT %MW1727 *)
    S102_M_DASH_PLT4_차종유 : BOOL; (* AT %MW1703.8 *)
    S102_M_DASH_PLT4_차종코드 : WORD; (* AT %MW1719 *)
    S102_M_DASH_PLT4_파트무 : BOOL; (* AT %MW1703.4 *)
    S102_M_DASH_PLT4_파트유 : BOOL; (* AT %MW1703.3 *)
    전체_M_이상_리셋 : BOOL; (* AT %MW308.2 *) (* 전체 M 이상 리셋 *)
END_VAR
VAR
    INST : TON;
    INST1 : TON;
    INST10 : TON;
    INST11 : TON;
    INST2 : TON;
    INST3 : TON;
    INST4 : TON;
    INST5 : TON;
    INST6 : TON;
    INST7 : TON;
    INST8 : TON;
    INST9 : TON;
    R201_1_M_I_RB_PROG_NO : INT;
    _R101_1_RB_비교_PROG_NO : INT;
    _R101_1_RH_APRON_PLT1_카운터_RST완료 : BOOL;
    _R101_1_RH_APRON_PLT1_카운터_RST요구 : BOOL;
    _R101_1_RH_APRON_PLT2_카운터_RST완료 : BOOL;
    _R101_1_RH_APRON_PLT2_카운터_RST요구 : BOOL;
    _R101_1_RH_PLT1_막장취출완료 : BOOL;
    _R101_1_RH_PLT2_막장취출완료 : BOOL;
    _R101_1_RH_PLT3_막장취출완료 : BOOL;
    _R101_1_RH_PLT4_막장취출완료 : BOOL;
    _R102_1_1_DASH_PLT1_카운터_RST완료 : BOOL;
    _R102_1_1_DASH_PLT1_카운터_RST요구 : BOOL;
    _R102_1_1_DASH_PLT2_카운터_RST완료 : BOOL;
    _R102_1_1_DASH_PLT2_카운터_RST요구 : BOOL;
    _R102_1_1_DASH_PLT3_카운터_RST완료 : BOOL;
    _R102_1_1_DASH_PLT3_카운터_RST요구 : BOOL;
    _R102_1_1_DASH_PLT4_카운터_RST완료 : BOOL;
    _R102_1_1_DASH_PLT4_카운터_RST요구 : BOOL;
    _R102_1_1_RB_비교_PROG_NO : INT;
    _R201_1_OTR_PLT1_카운터_RST완료 : BOOL;
    _R201_1_OTR_PLT1_카운터_RST요구 : BOOL;
    _R201_1_OTR_PLT2_카운터_RST완료 : BOOL;
    _R201_1_OTR_PLT2_카운터_RST요구 : BOOL;
    _R201_1_PLT1_막장취출완료 : BOOL;
    _R201_1_PLT2_막장취출완료 : BOOL;
    _R201_1_RB_비교_PROG_NO : INT;
    _R201_1_RB_비교_PROG_NO_INT : INT;
    _R201_1_막장취출완료 : BOOL;
    _랙1_제품수량 : INT;
    _랙1_차종코드 : INT;
    _랙2_제품수량 : INT;
    _랙2_차종코드 : INT;
END_VAR
VAR
    _p1 : BOOL;
    _p2 : BOOL;
    _p3 : BOOL;
    _p4 : BOOL;
END_VAR

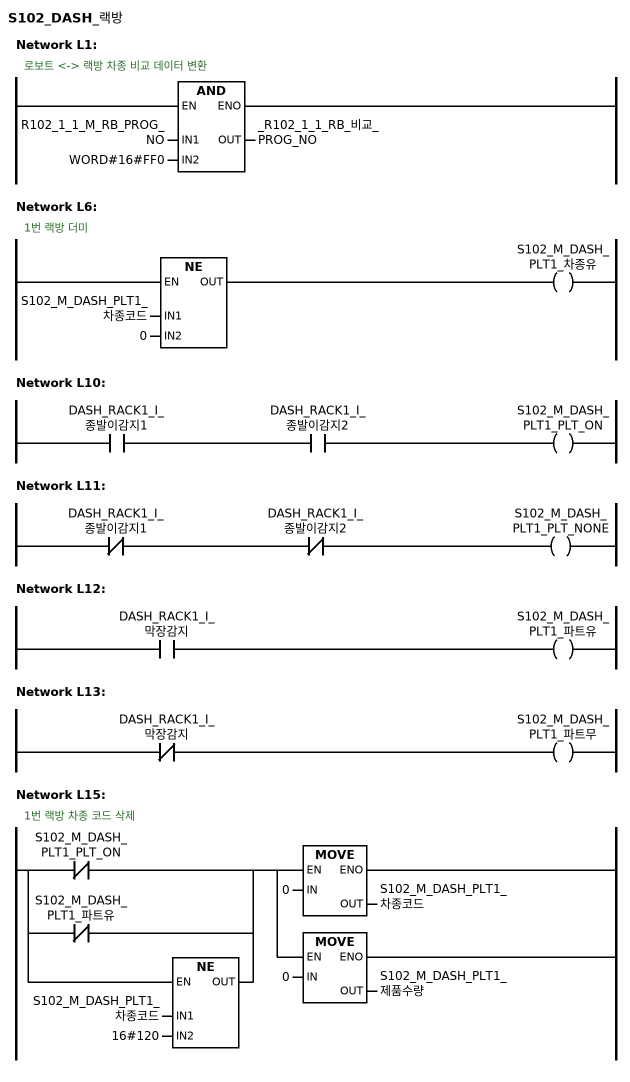
(* 로보트 <-> 랙방 차종 비교 데이터 변환 *)
(* Rung L1 *)
_R102_1_1_RB_비교_PROG_NO := R102_1_1_M_RB_PROG_NO AND WORD#16#FF0;
(* 1번 랙방 더미 *)
(* Rung L6 *)
S102_M_DASH_PLT1_차종유 := S102_M_DASH_PLT1_차종코드 <> 0;
(* Rung L10 *)
S102_M_DASH_PLT1_PLT_ON := DASH_RACK1_I_종발이감지1 AND DASH_RACK1_I_종발이감지2;
(* Rung L11 *)
S102_M_DASH_PLT1_PLT_NONE := NOT DASH_RACK1_I_종발이감지1 AND NOT DASH_RACK1_I_종발이감지2;
(* Rung L12 *)
S102_M_DASH_PLT1_파트유 := DASH_RACK1_I_막장감지;
(* Rung L13 *)
S102_M_DASH_PLT1_파트무 := NOT DASH_RACK1_I_막장감지;
(* 1번 랙방 차종 코드 삭제 *)
(* Rung L15 *)
_p1 := NOT S102_M_DASH_PLT1_PLT_ON OR NOT S102_M_DASH_PLT1_파트유 OR (S102_M_DASH_PLT1_차종코드 <> 16#120);
IF _p1 THEN
    S102_M_DASH_PLT1_차종코드 := 0;
    S102_M_DASH_PLT1_제품수량 := 0;
END_IF;
(* 1번 랙방 차종 코드 입력 *)
(* Rung L22: network not rendered *)
(* not connected or not rendered: S102_M_DASH_PLT1_로딩완료, S102_M_DASH_PLT1_PLT_ON, S102_M_DASH_PLT1_파트유, 16#120, S102_M_DASH_PLT1_차종코드, 10, S102_M_DASH_PLT1_제품수량 *)

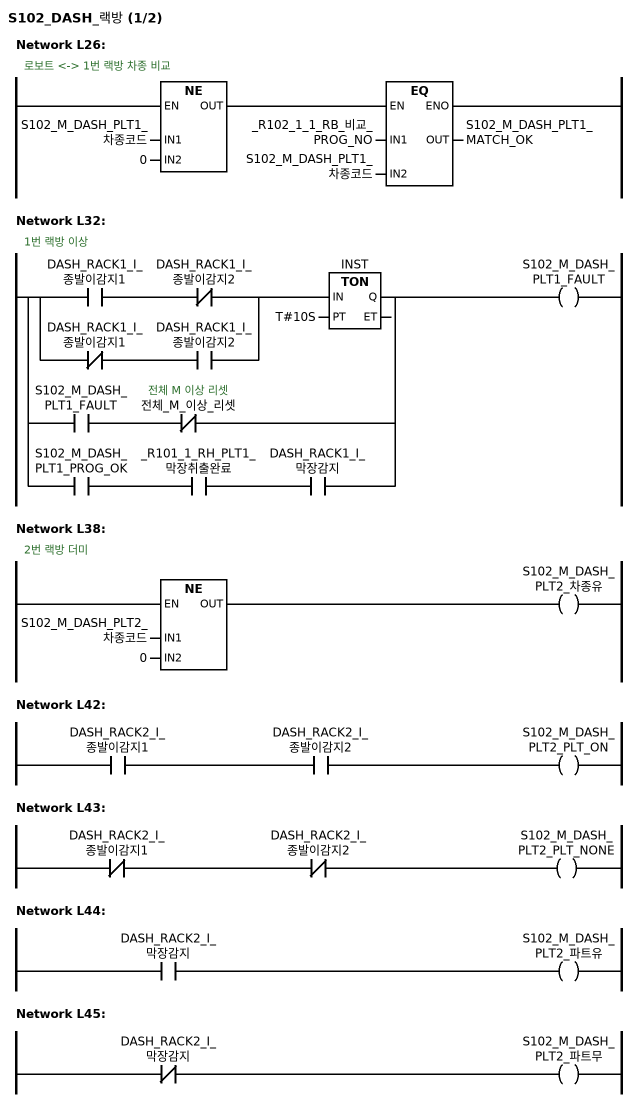
(* 로보트 <-> 1번 랙방 차종 비교 *)
(* Rung L26 *)
IF S102_M_DASH_PLT1_차종코드 <> 0 THEN
    S102_M_DASH_PLT1_MATCH_OK := _R102_1_1_RB_비교_PROG_NO = S102_M_DASH_PLT1_차종코드;
END_IF;
(* 1번 랙방 이상 *)
(* Rung L32 *)
INST(IN := (DASH_RACK1_I_종발이감지1 AND NOT DASH_RACK1_I_종발이감지2) OR (NOT DASH_RACK1_I_종발이감지1 AND DASH_RACK1_I_종발이감지2), PT := T#10S);
S102_M_DASH_PLT1_FAULT := INST.Q OR (S102_M_DASH_PLT1_FAULT AND NOT 전체_M_이상_리셋) OR (S102_M_DASH_PLT1_PROG_OK AND _R101_1_RH_PLT1_막장취출완료 AND DASH_RACK1_I_막장감지);
(* 2번 랙방 더미 *)
(* Rung L38 *)
S102_M_DASH_PLT2_차종유 := S102_M_DASH_PLT2_차종코드 <> 0;
(* Rung L42 *)
S102_M_DASH_PLT2_PLT_ON := DASH_RACK2_I_종발이감지1 AND DASH_RACK2_I_종발이감지2;
(* Rung L43 *)
S102_M_DASH_PLT2_PLT_NONE := NOT DASH_RACK2_I_종발이감지1 AND NOT DASH_RACK2_I_종발이감지2;
(* Rung L44 *)
S102_M_DASH_PLT2_파트유 := DASH_RACK2_I_막장감지;
(* Rung L45 *)
S102_M_DASH_PLT2_파트무 := NOT DASH_RACK2_I_막장감지;

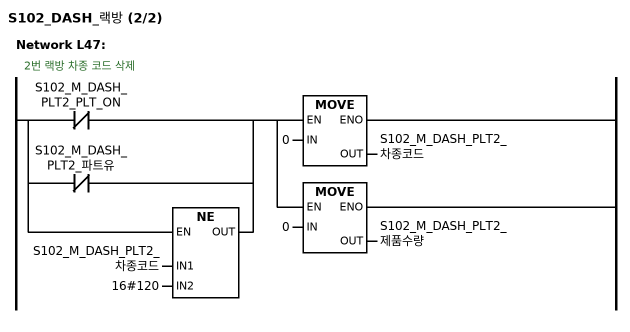
(* 2번 랙방 차종 코드 삭제 *)
(* Rung L47 *)
_p2 := NOT S102_M_DASH_PLT2_PLT_ON OR NOT S102_M_DASH_PLT2_파트유 OR (S102_M_DASH_PLT2_차종코드 <> 16#120);
IF _p2 THEN
    S102_M_DASH_PLT2_차종코드 := 0;
    S102_M_DASH_PLT2_제품수량 := 0;
END_IF;
(* 2번 랙방 차종 코드 입력 *)
(* Rung L54: network not rendered *)
(* not connected or not rendered: S102_M_DASH_PLT2_로딩완료, S102_M_DASH_PLT2_PLT_ON, S102_M_DASH_PLT2_파트유, 16#120, S102_M_DASH_PLT2_차종코드, 10, S102_M_DASH_PLT2_제품수량 *)

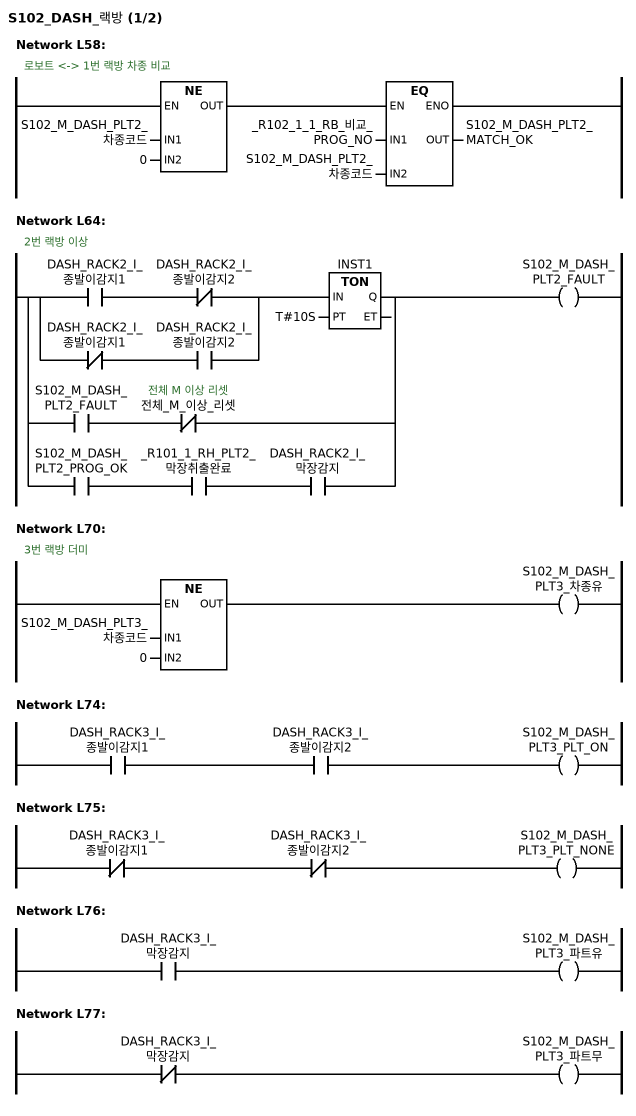
(* 로보트 <-> 1번 랙방 차종 비교 *)
(* Rung L58 *)
IF S102_M_DASH_PLT2_차종코드 <> 0 THEN
    S102_M_DASH_PLT2_MATCH_OK := _R102_1_1_RB_비교_PROG_NO = S102_M_DASH_PLT2_차종코드;
END_IF;
(* 2번 랙방 이상 *)
(* Rung L64 *)
INST1(IN := (DASH_RACK2_I_종발이감지1 AND NOT DASH_RACK2_I_종발이감지2) OR (NOT DASH_RACK2_I_종발이감지1 AND DASH_RACK2_I_종발이감지2), PT := T#10S);
S102_M_DASH_PLT2_FAULT := INST1.Q OR (S102_M_DASH_PLT2_FAULT AND NOT 전체_M_이상_리셋) OR (S102_M_DASH_PLT2_PROG_OK AND _R101_1_RH_PLT2_막장취출완료 AND DASH_RACK2_I_막장감지);
(* 3번 랙방 더미 *)
(* Rung L70 *)
S102_M_DASH_PLT3_차종유 := S102_M_DASH_PLT3_차종코드 <> 0;
(* Rung L74 *)
S102_M_DASH_PLT3_PLT_ON := DASH_RACK3_I_종발이감지1 AND DASH_RACK3_I_종발이감지2;
(* Rung L75 *)
S102_M_DASH_PLT3_PLT_NONE := NOT DASH_RACK3_I_종발이감지1 AND NOT DASH_RACK3_I_종발이감지2;
(* Rung L76 *)
S102_M_DASH_PLT3_파트유 := DASH_RACK3_I_막장감지;
(* Rung L77 *)
S102_M_DASH_PLT3_파트무 := NOT DASH_RACK3_I_막장감지;

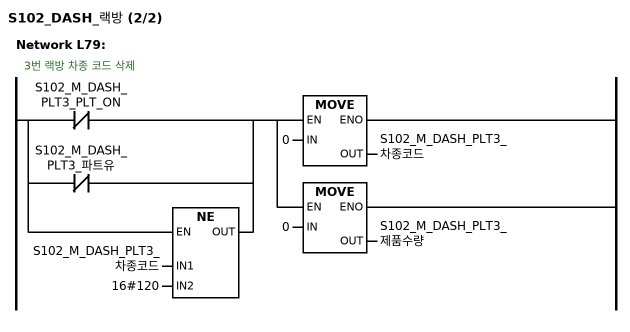
(* 3번 랙방 차종 코드 삭제 *)
(* Rung L79 *)
_p3 := NOT S102_M_DASH_PLT3_PLT_ON OR NOT S102_M_DASH_PLT3_파트유 OR (S102_M_DASH_PLT3_차종코드 <> 16#120);
IF _p3 THEN
    S102_M_DASH_PLT3_차종코드 := 0;
    S102_M_DASH_PLT3_제품수량 := 0;
END_IF;
(* 3번 랙방 차종 코드 입력 *)
(* Rung L86: network not rendered *)
(* not connected or not rendered: S102_M_DASH_PLT3_로딩완료, S102_M_DASH_PLT3_PLT_ON, S102_M_DASH_PLT3_파트유, 16#120, S102_M_DASH_PLT3_차종코드, 10, S102_M_DASH_PLT3_제품수량 *)

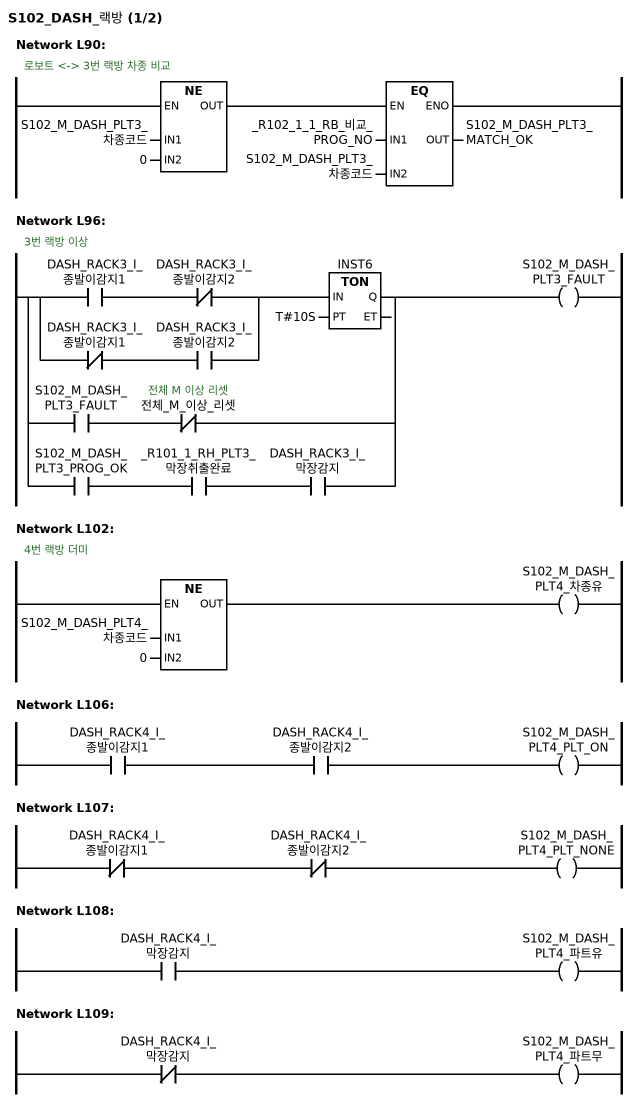
(* 로보트 <-> 3번 랙방 차종 비교 *)
(* Rung L90 *)
IF S102_M_DASH_PLT3_차종코드 <> 0 THEN
    S102_M_DASH_PLT3_MATCH_OK := _R102_1_1_RB_비교_PROG_NO = S102_M_DASH_PLT3_차종코드;
END_IF;
(* 3번 랙방 이상 *)
(* Rung L96 *)
INST6(IN := (DASH_RACK3_I_종발이감지1 AND NOT DASH_RACK3_I_종발이감지2) OR (NOT DASH_RACK3_I_종발이감지1 AND DASH_RACK3_I_종발이감지2), PT := T#10S);
S102_M_DASH_PLT3_FAULT := INST6.Q OR (S102_M_DASH_PLT3_FAULT AND NOT 전체_M_이상_리셋) OR (S102_M_DASH_PLT3_PROG_OK AND _R101_1_RH_PLT3_막장취출완료 AND DASH_RACK3_I_막장감지);
(* 4번 랙방 더미 *)
(* Rung L102 *)
S102_M_DASH_PLT4_차종유 := S102_M_DASH_PLT4_차종코드 <> 0;
(* Rung L106 *)
S102_M_DASH_PLT4_PLT_ON := DASH_RACK4_I_종발이감지1 AND DASH_RACK4_I_종발이감지2;
(* Rung L107 *)
S102_M_DASH_PLT4_PLT_NONE := NOT DASH_RACK4_I_종발이감지1 AND NOT DASH_RACK4_I_종발이감지2;
(* Rung L108 *)
S102_M_DASH_PLT4_파트유 := DASH_RACK4_I_막장감지;
(* Rung L109 *)
S102_M_DASH_PLT4_파트무 := NOT DASH_RACK4_I_막장감지;

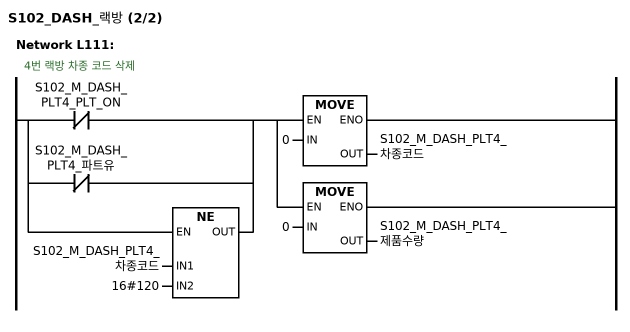
(* 4번 랙방 차종 코드 삭제 *)
(* Rung L111 *)
_p4 := NOT S102_M_DASH_PLT4_PLT_ON OR NOT S102_M_DASH_PLT4_파트유 OR (S102_M_DASH_PLT4_차종코드 <> 16#120);
IF _p4 THEN
    S102_M_DASH_PLT4_차종코드 := 0;
    S102_M_DASH_PLT4_제품수량 := 0;
END_IF;
(* 4번 랙방 차종 코드 입력 *)
(* Rung L118: network not rendered *)
(* not connected or not rendered: S102_M_DASH_PLT4_로딩완료, S102_M_DASH_PLT4_PLT_ON, S102_M_DASH_PLT4_파트유, 16#120, S102_M_DASH_PLT4_차종코드, 10, S102_M_DASH_PLT4_제품수량 *)

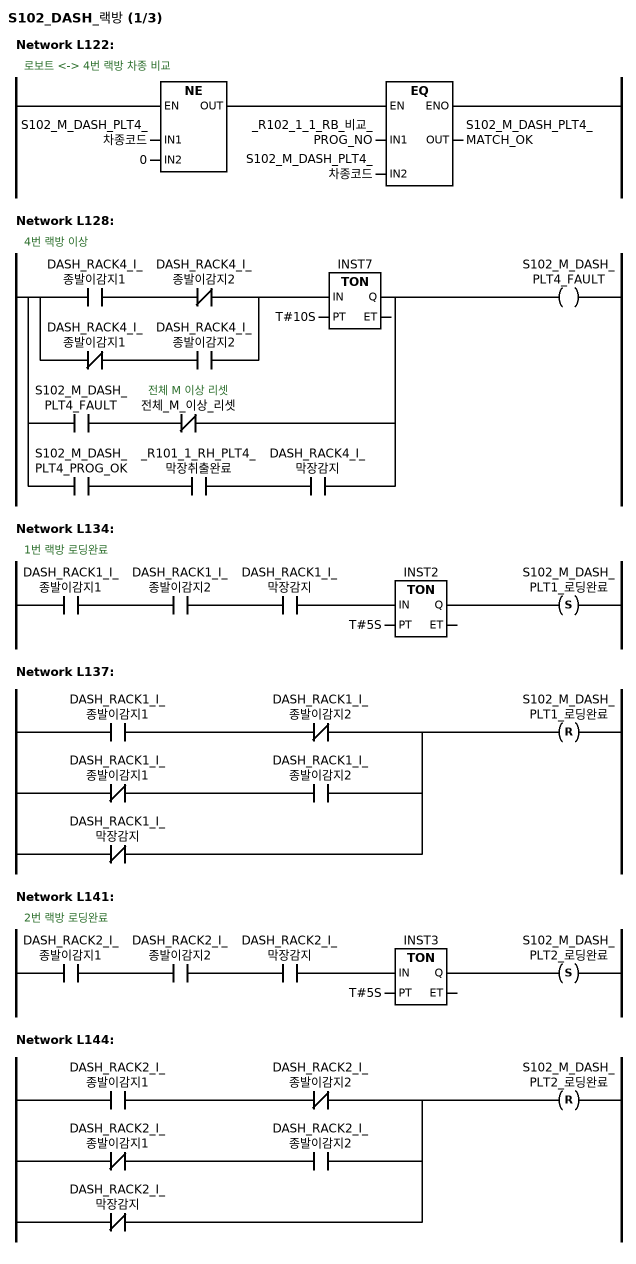
(* 로보트 <-> 4번 랙방 차종 비교 *)
(* Rung L122 *)
IF S102_M_DASH_PLT4_차종코드 <> 0 THEN
    S102_M_DASH_PLT4_MATCH_OK := _R102_1_1_RB_비교_PROG_NO = S102_M_DASH_PLT4_차종코드;
END_IF;
(* 4번 랙방 이상 *)
(* Rung L128 *)
INST7(IN := (DASH_RACK4_I_종발이감지1 AND NOT DASH_RACK4_I_종발이감지2) OR (NOT DASH_RACK4_I_종발이감지1 AND DASH_RACK4_I_종발이감지2), PT := T#10S);
S102_M_DASH_PLT4_FAULT := INST7.Q OR (S102_M_DASH_PLT4_FAULT AND NOT 전체_M_이상_리셋) OR (S102_M_DASH_PLT4_PROG_OK AND _R101_1_RH_PLT4_막장취출완료 AND DASH_RACK4_I_막장감지);
(* 1번 랙방 로딩완료 *)
(* Rung L134 *)
INST2(IN := DASH_RACK1_I_종발이감지1 AND DASH_RACK1_I_종발이감지2 AND DASH_RACK1_I_막장감지, PT := T#5S);
IF INST2.Q THEN S102_M_DASH_PLT1_로딩완료 := TRUE; END_IF;
(* Rung L137 *)
IF (DASH_RACK1_I_종발이감지1 AND NOT DASH_RACK1_I_종발이감지2) OR (NOT DASH_RACK1_I_종발이감지1 AND DASH_RACK1_I_종발이감지2) OR NOT DASH_RACK1_I_막장감지 THEN
    S102_M_DASH_PLT1_로딩완료 := FALSE;
END_IF;
(* 2번 랙방 로딩완료 *)
(* Rung L141 *)
INST3(IN := DASH_RACK2_I_종발이감지1 AND DASH_RACK2_I_종발이감지2 AND DASH_RACK2_I_막장감지, PT := T#5S);
IF INST3.Q THEN S102_M_DASH_PLT2_로딩완료 := TRUE; END_IF;
(* Rung L144 *)
IF (DASH_RACK2_I_종발이감지1 AND NOT DASH_RACK2_I_종발이감지2) OR (NOT DASH_RACK2_I_종발이감지1 AND DASH_RACK2_I_종발이감지2) OR NOT DASH_RACK2_I_막장감지 THEN
    S102_M_DASH_PLT2_로딩완료 := FALSE;
END_IF;

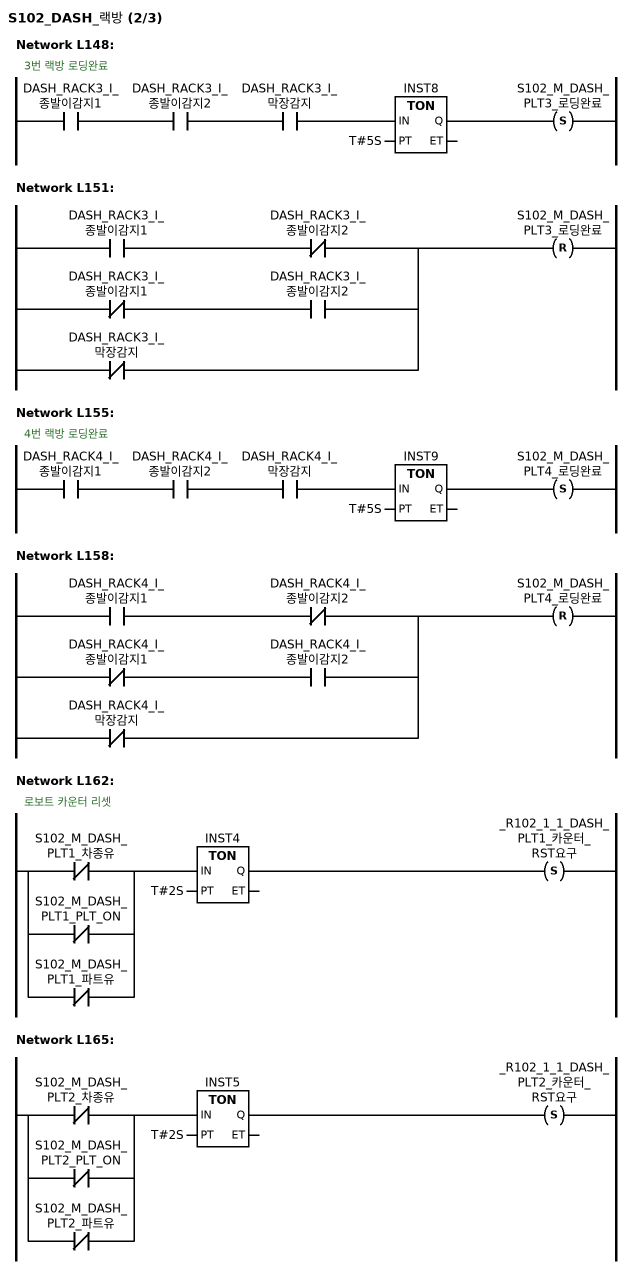
(* 3번 랙방 로딩완료 *)
(* Rung L148 *)
INST8(IN := DASH_RACK3_I_종발이감지1 AND DASH_RACK3_I_종발이감지2 AND DASH_RACK3_I_막장감지, PT := T#5S);
IF INST8.Q THEN S102_M_DASH_PLT3_로딩완료 := TRUE; END_IF;
(* Rung L151 *)
IF (DASH_RACK3_I_종발이감지1 AND NOT DASH_RACK3_I_종발이감지2) OR (NOT DASH_RACK3_I_종발이감지1 AND DASH_RACK3_I_종발이감지2) OR NOT DASH_RACK3_I_막장감지 THEN
    S102_M_DASH_PLT3_로딩완료 := FALSE;
END_IF;
(* 4번 랙방 로딩완료 *)
(* Rung L155 *)
INST9(IN := DASH_RACK4_I_종발이감지1 AND DASH_RACK4_I_종발이감지2 AND DASH_RACK4_I_막장감지, PT := T#5S);
IF INST9.Q THEN S102_M_DASH_PLT4_로딩완료 := TRUE; END_IF;
(* Rung L158 *)
IF (DASH_RACK4_I_종발이감지1 AND NOT DASH_RACK4_I_종발이감지2) OR (NOT DASH_RACK4_I_종발이감지1 AND DASH_RACK4_I_종발이감지2) OR NOT DASH_RACK4_I_막장감지 THEN
    S102_M_DASH_PLT4_로딩완료 := FALSE;
END_IF;
(* 로보트 카운터 리셋 *)
(* Rung L162 *)
INST4(IN := NOT S102_M_DASH_PLT1_차종유 OR NOT S102_M_DASH_PLT1_PLT_ON OR NOT S102_M_DASH_PLT1_파트유, PT := T#2S);
IF INST4.Q THEN _R102_1_1_DASH_PLT1_카운터_RST요구 := TRUE; END_IF;
(* Rung L165 *)
INST5(IN := NOT S102_M_DASH_PLT2_차종유 OR NOT S102_M_DASH_PLT2_PLT_ON OR NOT S102_M_DASH_PLT2_파트유, PT := T#2S);
IF INST5.Q THEN _R102_1_1_DASH_PLT2_카운터_RST요구 := TRUE; END_IF;

